(* Logix 5000 project; controller AMANA_DC_PLANT_01 vendor 1 type 14 code 164 rev 31.12; software revision 31.02 *)

TASK MainTask (continuous, watchdog 500 ms) : LN00, OH_BARCODE_SCAN

MODULES
   Local : vendor 1 type 14 code 164 (ICP 0, rev 31.12)
      EN4TR : 1756-EN4TR (ICP 3, Ethernet 192.168.1.1, rev 2.1, Input RPI 500 ms)
         Test_ArmorBlock : vendor 1 type 7 code 357 (Ethernet 192.168.1.100, rev 1.1, Output RPI 20 ms)
      OH_SCAN_DOCKSORTING : SR-2000 (Ethernet 10.28.17.144, rev 1.1, StandardDataDriven RPI 20 ms)
           OH_SCAN_DOCKSORTING:I.Data[0].0   // Error
           OH_SCAN_DOCKSORTING:I.Data[0].1   // Result Data Available
           OH_SCAN_DOCKSORTING:I.Data[0].2   // Result Data Strobe
           OH_SCAN_DOCKSORTING:I.Data[0].3   // Reserved
           OH_SCAN_DOCKSORTING:I.Data[0].4   // Reserved
           OH_SCAN_DOCKSORTING:I.Data[0].5   // Reserved
           OH_SCAN_DOCKSORTING:I.Data[0].6   // Buffer Overflow Error
           OH_SCAN_DOCKSORTING:I.Data[0].7   // General Error
           OH_SCAN_DOCKSORTING:I.Data[10]   // ISO/IEC15415 Grade
           OH_SCAN_DOCKSORTING:I.Data[11]   // Reserved
           OH_SCAN_DOCKSORTING:I.Data[12]   // AIM DPM Grade
           OH_SCAN_DOCKSORTING:I.Data[13]   // Reserved
           OH_SCAN_DOCKSORTING:I.Data[14]   // ISO/IEC15416 Grade
           OH_SCAN_DOCKSORTING:I.Data[15]   // Reserved
           OH_SCAN_DOCKSORTING:I.Data[16]   // Read Result Code
           OH_SCAN_DOCKSORTING:I.Data[17]   // Read Result Code
           OH_SCAN_DOCKSORTING:I.Data[18]   // Preset Result Code
           OH_SCAN_DOCKSORTING:I.Data[19]   // Preset Result Code
           OH_SCAN_DOCKSORTING:I.Data[1].0   // Busy
           OH_SCAN_DOCKSORTING:I.Data[1].1   // Trigger Busy
           OH_SCAN_DOCKSORTING:I.Data[1].2   // Lock Busy
           OH_SCAN_DOCKSORTING:I.Data[1].3   // Mode Busy
           OH_SCAN_DOCKSORTING:I.Data[1].4   // Error Busy
           OH_SCAN_DOCKSORTING:I.Data[1].5   // Reserved
           OH_SCAN_DOCKSORTING:I.Data[1].6   // Ready
           OH_SCAN_DOCKSORTING:I.Data[1].7   // Reserved
           OH_SCAN_DOCKSORTING:I.Data[20]   // Register Preset Data Result Code
           OH_SCAN_DOCKSORTING:I.Data[21]   // Register Preset Data Result Code
           OH_SCAN_DOCKSORTING:I.Data[22]   // Tune Result Code
           OH_SCAN_DOCKSORTING:I.Data[23]   // Tune Result Code
           OH_SCAN_DOCKSORTING:I.Data[24]   // Bload Result Code
           OH_SCAN_DOCKSORTING:I.Data[25]   // Bload Result Code
           OH_SCAN_DOCKSORTING:I.Data[26]   // Reserved
           OH_SCAN_DOCKSORTING:I.Data[27]   // Reserved
           OH_SCAN_DOCKSORTING:I.Data[28]   // Reserved
           OH_SCAN_DOCKSORTING:I.Data[29]   // Reserved
           OH_SCAN_DOCKSORTING:I.Data[2].0   // Read Complete
           OH_SCAN_DOCKSORTING:I.Data[2].1   // Preset Complete
           OH_SCAN_DOCKSORTING:I.Data[2].2   // Register Preset Data Complete
           OH_SCAN_DOCKSORTING:I.Data[2].3   // Tune Complete
           OH_SCAN_DOCKSORTING:I.Data[2].4   // Bload Complete
           OH_SCAN_DOCKSORTING:I.Data[2].5   // Reserved
           OH_SCAN_DOCKSORTING:I.Data[2].6   // Reserved
           OH_SCAN_DOCKSORTING:I.Data[2].7   // External Request Complete
           OH_SCAN_DOCKSORTING:I.Data[30]   // External Request Result Code
           OH_SCAN_DOCKSORTING:I.Data[31]   // External Request Result Code
           OH_SCAN_DOCKSORTING:I.Data[32]   // General Error Code
           OH_SCAN_DOCKSORTING:I.Data[33]   // General Error Code
           OH_SCAN_DOCKSORTING:I.Data[34]   // Slave ID
           OH_SCAN_DOCKSORTING:I.Data[35]   // Slave ID
           OH_SCAN_DOCKSORTING:I.Data[36]   // Result Data Ready Count
           OH_SCAN_DOCKSORTING:I.Data[37]   // Result Data Ready Count
           OH_SCAN_DOCKSORTING:I.Data[38]   // Result Data Update Count
           OH_SCAN_DOCKSORTING:I.Data[39]   // Result Data Update Count
           OH_SCAN_DOCKSORTING:I.Data[3].0   // Read Failure
           OH_SCAN_DOCKSORTING:I.Data[3].1   // Preset Failure
           OH_SCAN_DOCKSORTING:I.Data[3].2   // Register Preset Data Failure
           OH_SCAN_DOCKSORTING:I.Data[3].3   // Tune Failure
           OH_SCAN_DOCKSORTING:I.Data[3].4   // Bload Failure
           OH_SCAN_DOCKSORTING:I.Data[3].5   // Reserved
           OH_SCAN_DOCKSORTING:I.Data[3].6   // Reserved
           OH_SCAN_DOCKSORTING:I.Data[3].7   // External Request Failure
           OH_SCAN_DOCKSORTING:I.Data[40]   // Trigger Input Count for Master
           OH_SCAN_DOCKSORTING:I.Data[41]   // Trigger Input Count for Master
           OH_SCAN_DOCKSORTING:I.Data[42]   // Result Data Size
           OH_SCAN_DOCKSORTING:I.Data[43]   // Result Data Size
           OH_SCAN_DOCKSORTING:I.Data[44]   // Result Data
           OH_SCAN_DOCKSORTING:I.Data[45]   // Result Data
           OH_SCAN_DOCKSORTING:I.Data[46]   // Result Data
           OH_SCAN_DOCKSORTING:I.Data[47]   // Result Data
           OH_SCAN_DOCKSORTING:I.Data[48]   // Result Data
           OH_SCAN_DOCKSORTING:I.Data[49]   // Result Data
           OH_SCAN_DOCKSORTING:I.Data[4].0   // Input 1 Status
           OH_SCAN_DOCKSORTING:I.Data[4].1   // Input 2 Status
           OH_SCAN_DOCKSORTING:I.Data[4].2   // Reserved
           OH_SCAN_DOCKSORTING:I.Data[4].3   // Reserved
           OH_SCAN_DOCKSORTING:I.Data[4].4   // Output 1 Status
           OH_SCAN_DOCKSORTING:I.Data[4].5   // Output 2 Status
           OH_SCAN_DOCKSORTING:I.Data[4].6   // Output 3 Status
           OH_SCAN_DOCKSORTING:I.Data[4].7   // Reserved
           OH_SCAN_DOCKSORTING:I.Data[50]   // Result Data
           OH_SCAN_DOCKSORTING:I.Data[5].0   // Unstable
           OH_SCAN_DOCKSORTING:I.Data[5].1   // Matching Level Unstable
           OH_SCAN_DOCKSORTING:I.Data[5].2   // ISO/IEC15415 Unstable
           OH_SCAN_DOCKSORTING:I.Data[5].3   // AIM DPM Unstable
           OH_SCAN_DOCKSORTING:I.Data[5].4   // ADE AS9132 Unstable
           OH_SCAN_DOCKSORTING:I.Data[5].5   // ISO/IEC15416 Unstable
           OH_SCAN_DOCKSORTING:I.Data[5].6   // Reserved
           OH_SCAN_DOCKSORTING:I.Data[5].7   // Reserved
           OH_SCAN_DOCKSORTING:I.Data[6]   // Reserved
           OH_SCAN_DOCKSORTING:I.Data[7]   // Reserved
           OH_SCAN_DOCKSORTING:I.Data[8]   // Matching Level
           OH_SCAN_DOCKSORTING:I.Data[9]   // Reserved
           OH_SCAN_DOCKSORTING:O.Data[0].0   // Reserved
           OH_SCAN_DOCKSORTING:O.Data[0].1   // Result Data Latch
           OH_SCAN_DOCKSORTING:O.Data[0].2   // Reserved
           OH_SCAN_DOCKSORTING:O.Data[0].3   // Reserved
           OH_SCAN_DOCKSORTING:O.Data[0].4   // Reserved
           OH_SCAN_DOCKSORTING:O.Data[0].5   // Reserved
           OH_SCAN_DOCKSORTING:O.Data[0].6   // Reserved
           OH_SCAN_DOCKSORTING:O.Data[0].7   // Error Clear
           OH_SCAN_DOCKSORTING:O.Data[10]   // User Data Size
           OH_SCAN_DOCKSORTING:O.Data[11]   // User Data Size
           OH_SCAN_DOCKSORTING:O.Data[12]   // User Data
           OH_SCAN_DOCKSORTING:O.Data[13]   // User Data
           OH_SCAN_DOCKSORTING:O.Data[14]   // User Data
           OH_SCAN_DOCKSORTING:O.Data[15]   // User Data
           OH_SCAN_DOCKSORTING:O.Data[16]   // User Data
           OH_SCAN_DOCKSORTING:O.Data[17]   // User Data
           OH_SCAN_DOCKSORTING:O.Data[1].0   // Read Request
           OH_SCAN_DOCKSORTING:O.Data[1].1   // Preset Request
           OH_SCAN_DOCKSORTING:O.Data[1].2   // Register Preset Data Request
           OH_SCAN_DOCKSORTING:O.Data[1].3   // Tune Request
           OH_SCAN_DOCKSORTING:O.Data[1].4   // Bload Request
           OH_SCAN_DOCKSORTING:O.Data[1].5   // Reserved
           OH_SCAN_DOCKSORTING:O.Data[1].6   // Reserved
           OH_SCAN_DOCKSORTING:O.Data[1].7   // Reserved
           OH_SCAN_DOCKSORTING:O.Data[2].0   // Read Complete Clear
           OH_SCAN_DOCKSORTING:O.Data[2].1   // Preset Complete Clear
           OH_SCAN_DOCKSORTING:O.Data[2].2   // Register Preset Data Complete Clear
           OH_SCAN_DOCKSORTING:O.Data[2].3   // Tune Complete Clear
           OH_SCAN_DOCKSORTING:O.Data[2].4   // Bload Complete Clear
           OH_SCAN_DOCKSORTING:O.Data[2].5   // Reserved
           OH_SCAN_DOCKSORTING:O.Data[2].6   // Reserved
           OH_SCAN_DOCKSORTING:O.Data[2].7   // External Request Complete Clear
           OH_SCAN_DOCKSORTING:O.Data[3]   // Reserved
           OH_SCAN_DOCKSORTING:O.Data[4]   // Bank Number
           OH_SCAN_DOCKSORTING:O.Data[5]   // Bank Number
           OH_SCAN_DOCKSORTING:O.Data[6]   // Reserved
           OH_SCAN_DOCKSORTING:O.Data[7]   // Reserved
           OH_SCAN_DOCKSORTING:O.Data[8]   // Reserved
           OH_SCAN_DOCKSORTING:O.Data[9]   // Reserved
      OH_SCAN_WAREHOUSENORTH : SR-2000 (Ethernet 10.28.17.138, rev 1.1, StandardDataDriven RPI 20 ms)
           OH_SCAN_WAREHOUSENORTH:I.Data[0].0   // Error
           OH_SCAN_WAREHOUSENORTH:I.Data[0].1   // Result Data Available
           OH_SCAN_WAREHOUSENORTH:I.Data[0].2   // Result Data Strobe
           OH_SCAN_WAREHOUSENORTH:I.Data[0].3   // Reserved
           OH_SCAN_WAREHOUSENORTH:I.Data[0].4   // Reserved
           OH_SCAN_WAREHOUSENORTH:I.Data[0].5   // Reserved
           OH_SCAN_WAREHOUSENORTH:I.Data[0].6   // Buffer Overflow Error
           OH_SCAN_WAREHOUSENORTH:I.Data[0].7   // General Error
           OH_SCAN_WAREHOUSENORTH:I.Data[10]   // ISO/IEC15415 Grade
           OH_SCAN_WAREHOUSENORTH:I.Data[11]   // Reserved
           OH_SCAN_WAREHOUSENORTH:I.Data[12]   // AIM DPM Grade
           OH_SCAN_WAREHOUSENORTH:I.Data[13]   // Reserved
           OH_SCAN_WAREHOUSENORTH:I.Data[14]   // ISO/IEC15416 Grade
           OH_SCAN_WAREHOUSENORTH:I.Data[15]   // Reserved
           OH_SCAN_WAREHOUSENORTH:I.Data[16]   // Read Result Code
           OH_SCAN_WAREHOUSENORTH:I.Data[17]   // Read Result Code
           OH_SCAN_WAREHOUSENORTH:I.Data[18]   // Preset Result Code
           OH_SCAN_WAREHOUSENORTH:I.Data[19]   // Preset Result Code
           OH_SCAN_WAREHOUSENORTH:I.Data[1].0   // Busy
           OH_SCAN_WAREHOUSENORTH:I.Data[1].1   // Trigger Busy
           OH_SCAN_WAREHOUSENORTH:I.Data[1].2   // Lock Busy
           OH_SCAN_WAREHOUSENORTH:I.Data[1].3   // Mode Busy
           OH_SCAN_WAREHOUSENORTH:I.Data[1].4   // Error Busy
           OH_SCAN_WAREHOUSENORTH:I.Data[1].5   // Reserved
           OH_SCAN_WAREHOUSENORTH:I.Data[1].6   // Ready
           OH_SCAN_WAREHOUSENORTH:I.Data[1].7   // Reserved
           OH_SCAN_WAREHOUSENORTH:I.Data[20]   // Register Preset Data Result Code
           OH_SCAN_WAREHOUSENORTH:I.Data[21]   // Register Preset Data Result Code
           OH_SCAN_WAREHOUSENORTH:I.Data[22]   // Tune Result Code
           OH_SCAN_WAREHOUSENORTH:I.Data[23]   // Tune Result Code
           OH_SCAN_WAREHOUSENORTH:I.Data[24]   // Bload Result Code
           OH_SCAN_WAREHOUSENORTH:I.Data[25]   // Bload Result Code
           OH_SCAN_WAREHOUSENORTH:I.Data[26]   // Reserved
           OH_SCAN_WAREHOUSENORTH:I.Data[27]   // Reserved
           OH_SCAN_WAREHOUSENORTH:I.Data[28]   // Reserved
           OH_SCAN_WAREHOUSENORTH:I.Data[29]   // Reserved
           OH_SCAN_WAREHOUSENORTH:I.Data[2].0   // Read Complete
           OH_SCAN_WAREHOUSENORTH:I.Data[2].1   // Preset Complete
           OH_SCAN_WAREHOUSENORTH:I.Data[2].2   // Register Preset Data Complete
           OH_SCAN_WAREHOUSENORTH:I.Data[2].3   // Tune Complete
           OH_SCAN_WAREHOUSENORTH:I.Data[2].4   // Bload Complete
           OH_SCAN_WAREHOUSENORTH:I.Data[2].5   // Reserved
           OH_SCAN_WAREHOUSENORTH:I.Data[2].6   // Reserved
           OH_SCAN_WAREHOUSENORTH:I.Data[2].7   // External Request Complete
           OH_SCAN_WAREHOUSENORTH:I.Data[30]   // External Request Result Code
           OH_SCAN_WAREHOUSENORTH:I.Data[31]   // External Request Result Code
           OH_SCAN_WAREHOUSENORTH:I.Data[32]   // General Error Code
           OH_SCAN_WAREHOUSENORTH:I.Data[33]   // General Error Code
           OH_SCAN_WAREHOUSENORTH:I.Data[34]   // Slave ID
           OH_SCAN_WAREHOUSENORTH:I.Data[35]   // Slave ID
           OH_SCAN_WAREHOUSENORTH:I.Data[36]   // Result Data Ready Count
           OH_SCAN_WAREHOUSENORTH:I.Data[37]   // Result Data Ready Count
           OH_SCAN_WAREHOUSENORTH:I.Data[38]   // Result Data Update Count
           OH_SCAN_WAREHOUSENORTH:I.Data[39]   // Result Data Update Count
           OH_SCAN_WAREHOUSENORTH:I.Data[3].0   // Read Failure
           OH_SCAN_WAREHOUSENORTH:I.Data[3].1   // Preset Failure
           OH_SCAN_WAREHOUSENORTH:I.Data[3].2   // Register Preset Data Failure
           OH_SCAN_WAREHOUSENORTH:I.Data[3].3   // Tune Failure
           OH_SCAN_WAREHOUSENORTH:I.Data[3].4   // Bload Failure
           OH_SCAN_WAREHOUSENORTH:I.Data[3].5   // Reserved
           OH_SCAN_WAREHOUSENORTH:I.Data[3].6   // Reserved
           OH_SCAN_WAREHOUSENORTH:I.Data[3].7   // External Request Failure
           OH_SCAN_WAREHOUSENORTH:I.Data[40]   // Trigger Input Count for Master
           OH_SCAN_WAREHOUSENORTH:I.Data[41]   // Trigger Input Count for Master
           OH_SCAN_WAREHOUSENORTH:I.Data[42]   // Result Data Size
           OH_SCAN_WAREHOUSENORTH:I.Data[43]   // Result Data Size
           OH_SCAN_WAREHOUSENORTH:I.Data[44]   // Result Data
           OH_SCAN_WAREHOUSENORTH:I.Data[45]   // Result Data
           OH_SCAN_WAREHOUSENORTH:I.Data[46]   // Result Data
           OH_SCAN_WAREHOUSENORTH:I.Data[47]   // Result Data
           OH_SCAN_WAREHOUSENORTH:I.Data[48]   // Result Data
           OH_SCAN_WAREHOUSENORTH:I.Data[49]   // Result Data
           OH_SCAN_WAREHOUSENORTH:I.Data[4].0   // Input 1 Status
           OH_SCAN_WAREHOUSENORTH:I.Data[4].1   // Input 2 Status
           OH_SCAN_WAREHOUSENORTH:I.Data[4].2   // Reserved
           OH_SCAN_WAREHOUSENORTH:I.Data[4].3   // Reserved
           OH_SCAN_WAREHOUSENORTH:I.Data[4].4   // Output 1 Status
           OH_SCAN_WAREHOUSENORTH:I.Data[4].5   // Output 2 Status
           OH_SCAN_WAREHOUSENORTH:I.Data[4].6   // Output 3 Status
           OH_SCAN_WAREHOUSENORTH:I.Data[4].7   // Reserved
           OH_SCAN_WAREHOUSENORTH:I.Data[50]   // Result Data
           OH_SCAN_WAREHOUSENORTH:I.Data[5].0   // Unstable
           OH_SCAN_WAREHOUSENORTH:I.Data[5].1   // Matching Level Unstable
           OH_SCAN_WAREHOUSENORTH:I.Data[5].2   // ISO/IEC15415 Unstable
           OH_SCAN_WAREHOUSENORTH:I.Data[5].3   // AIM DPM Unstable
           OH_SCAN_WAREHOUSENORTH:I.Data[5].4   // ADE AS9132 Unstable
           OH_SCAN_WAREHOUSENORTH:I.Data[5].5   // ISO/IEC15416 Unstable
           OH_SCAN_WAREHOUSENORTH:I.Data[5].6   // Reserved
           OH_SCAN_WAREHOUSENORTH:I.Data[5].7   // Reserved
           OH_SCAN_WAREHOUSENORTH:I.Data[6]   // Reserved
           OH_SCAN_WAREHOUSENORTH:I.Data[7]   // Reserved
           OH_SCAN_WAREHOUSENORTH:I.Data[8]   // Matching Level
           OH_SCAN_WAREHOUSENORTH:I.Data[9]   // Reserved
           OH_SCAN_WAREHOUSENORTH:O.Data[0].0   // Reserved
           OH_SCAN_WAREHOUSENORTH:O.Data[0].1   // Result Data Latch
           OH_SCAN_WAREHOUSENORTH:O.Data[0].2   // Reserved
           OH_SCAN_WAREHOUSENORTH:O.Data[0].3   // Reserved
           OH_SCAN_WAREHOUSENORTH:O.Data[0].4   // Reserved
           OH_SCAN_WAREHOUSENORTH:O.Data[0].5   // Reserved
           OH_SCAN_WAREHOUSENORTH:O.Data[0].6   // Reserved
           OH_SCAN_WAREHOUSENORTH:O.Data[0].7   // Error Clear
           OH_SCAN_WAREHOUSENORTH:O.Data[10]   // User Data Size
           OH_SCAN_WAREHOUSENORTH:O.Data[11]   // User Data Size
           OH_SCAN_WAREHOUSENORTH:O.Data[12]   // User Data
           OH_SCAN_WAREHOUSENORTH:O.Data[13]   // User Data
           OH_SCAN_WAREHOUSENORTH:O.Data[14]   // User Data
           OH_SCAN_WAREHOUSENORTH:O.Data[15]   // User Data
           OH_SCAN_WAREHOUSENORTH:O.Data[16]   // User Data
           OH_SCAN_WAREHOUSENORTH:O.Data[17]   // User Data
           OH_SCAN_WAREHOUSENORTH:O.Data[1].0   // Read Request
           OH_SCAN_WAREHOUSENORTH:O.Data[1].1   // Preset Request
           OH_SCAN_WAREHOUSENORTH:O.Data[1].2   // Register Preset Data Request
           OH_SCAN_WAREHOUSENORTH:O.Data[1].3   // Tune Request
           OH_SCAN_WAREHOUSENORTH:O.Data[1].4   // Bload Request
           OH_SCAN_WAREHOUSENORTH:O.Data[1].5   // Reserved
           OH_SCAN_WAREHOUSENORTH:O.Data[1].6   // Reserved
           OH_SCAN_WAREHOUSENORTH:O.Data[1].7   // Reserved
           OH_SCAN_WAREHOUSENORTH:O.Data[2].0   // Read Complete Clear
           OH_SCAN_WAREHOUSENORTH:O.Data[2].1   // Preset Complete Clear
           OH_SCAN_WAREHOUSENORTH:O.Data[2].2   // Register Preset Data Complete Clear
           OH_SCAN_WAREHOUSENORTH:O.Data[2].3   // Tune Complete Clear
           OH_SCAN_WAREHOUSENORTH:O.Data[2].4   // Bload Complete Clear
           OH_SCAN_WAREHOUSENORTH:O.Data[2].5   // Reserved
           OH_SCAN_WAREHOUSENORTH:O.Data[2].6   // Reserved
           OH_SCAN_WAREHOUSENORTH:O.Data[2].7   // External Request Complete Clear
           OH_SCAN_WAREHOUSENORTH:O.Data[3]   // Reserved
           OH_SCAN_WAREHOUSENORTH:O.Data[4]   // Bank Number
           OH_SCAN_WAREHOUSENORTH:O.Data[5]   // Bank Number
           OH_SCAN_WAREHOUSENORTH:O.Data[6]   // Reserved
           OH_SCAN_WAREHOUSENORTH:O.Data[7]   // Reserved
           OH_SCAN_WAREHOUSENORTH:O.Data[8]   // Reserved
           OH_SCAN_WAREHOUSENORTH:O.Data[9]   // Reserved
      OH_SCAN_LN6 : SR-2000 (Ethernet 10.28.114.160, rev 1.1, StandardDataDriven RPI 20 ms)
           OH_SCAN_LN6:I.Data[0].0   // Error
           OH_SCAN_LN6:I.Data[0].1   // Result Data Available
           OH_SCAN_LN6:I.Data[0].2   // Result Data Strobe
           OH_SCAN_LN6:I.Data[0].3   // Reserved
           OH_SCAN_LN6:I.Data[0].4   // Reserved
           OH_SCAN_LN6:I.Data[0].5   // Reserved
           OH_SCAN_LN6:I.Data[0].6   // Buffer Overflow Error
           OH_SCAN_LN6:I.Data[0].7   // General Error
           OH_SCAN_LN6:I.Data[10]   // ISO/IEC15415 Grade
           OH_SCAN_LN6:I.Data[11]   // Reserved
           OH_SCAN_LN6:I.Data[12]   // AIM DPM Grade
           OH_SCAN_LN6:I.Data[13]   // Reserved
           OH_SCAN_LN6:I.Data[14]   // ISO/IEC15416 Grade
           OH_SCAN_LN6:I.Data[15]   // Reserved
           OH_SCAN_LN6:I.Data[16]   // Read Result Code
           OH_SCAN_LN6:I.Data[17]   // Read Result Code
           OH_SCAN_LN6:I.Data[18]   // Preset Result Code
           OH_SCAN_LN6:I.Data[19]   // Preset Result Code
           OH_SCAN_LN6:I.Data[1].0   // Busy
           OH_SCAN_LN6:I.Data[1].1   // Trigger Busy
           OH_SCAN_LN6:I.Data[1].2   // Lock Busy
           OH_SCAN_LN6:I.Data[1].3   // Mode Busy
           OH_SCAN_LN6:I.Data[1].4   // Error Busy
           OH_SCAN_LN6:I.Data[1].5   // Reserved
           OH_SCAN_LN6:I.Data[1].6   // Ready
           OH_SCAN_LN6:I.Data[1].7   // Reserved
           OH_SCAN_LN6:I.Data[20]   // Register Preset Data Result Code
           OH_SCAN_LN6:I.Data[21]   // Register Preset Data Result Code
           OH_SCAN_LN6:I.Data[22]   // Tune Result Code
           OH_SCAN_LN6:I.Data[23]   // Tune Result Code
           OH_SCAN_LN6:I.Data[24]   // Bload Result Code
           OH_SCAN_LN6:I.Data[25]   // Bload Result Code
           OH_SCAN_LN6:I.Data[26]   // Reserved
           OH_SCAN_LN6:I.Data[27]   // Reserved
           OH_SCAN_LN6:I.Data[28]   // Reserved
           OH_SCAN_LN6:I.Data[29]   // Reserved
           OH_SCAN_LN6:I.Data[2].0   // Read Complete
           OH_SCAN_LN6:I.Data[2].1   // Preset Complete
           OH_SCAN_LN6:I.Data[2].2   // Register Preset Data Complete
           OH_SCAN_LN6:I.Data[2].3   // Tune Complete
           OH_SCAN_LN6:I.Data[2].4   // Bload Complete
           OH_SCAN_LN6:I.Data[2].5   // Reserved
           OH_SCAN_LN6:I.Data[2].6   // Reserved
           OH_SCAN_LN6:I.Data[2].7   // External Request Complete
           OH_SCAN_LN6:I.Data[30]   // External Request Result Code
           OH_SCAN_LN6:I.Data[31]   // External Request Result Code
           OH_SCAN_LN6:I.Data[32]   // General Error Code
           OH_SCAN_LN6:I.Data[33]   // General Error Code
           OH_SCAN_LN6:I.Data[34]   // Slave ID
           OH_SCAN_LN6:I.Data[35]   // Slave ID
           OH_SCAN_LN6:I.Data[36]   // Result Data Ready Count
           OH_SCAN_LN6:I.Data[37]   // Result Data Ready Count
           OH_SCAN_LN6:I.Data[38]   // Result Data Update Count
           OH_SCAN_LN6:I.Data[39]   // Result Data Update Count
           OH_SCAN_LN6:I.Data[3].0   // Read Failure
           OH_SCAN_LN6:I.Data[3].1   // Preset Failure
           OH_SCAN_LN6:I.Data[3].2   // Register Preset Data Failure
           OH_SCAN_LN6:I.Data[3].3   // Tune Failure
           OH_SCAN_LN6:I.Data[3].4   // Bload Failure
           OH_SCAN_LN6:I.Data[3].5   // Reserved
           OH_SCAN_LN6:I.Data[3].6   // Reserved
           OH_SCAN_LN6:I.Data[3].7   // External Request Failure
           OH_SCAN_LN6:I.Data[40]   // Trigger Input Count for Master
           OH_SCAN_LN6:I.Data[41]   // Trigger Input Count for Master
           OH_SCAN_LN6:I.Data[42]   // Result Data Size
           OH_SCAN_LN6:I.Data[43]   // Result Data Size
           OH_SCAN_LN6:I.Data[44]   // Result Data
           OH_SCAN_LN6:I.Data[45]   // Result Data
           OH_SCAN_LN6:I.Data[46]   // Result Data
           OH_SCAN_LN6:I.Data[47]   // Result Data
           OH_SCAN_LN6:I.Data[48]   // Result Data
           OH_SCAN_LN6:I.Data[49]   // Result Data
           OH_SCAN_LN6:I.Data[4].0   // Input 1 Status
           OH_SCAN_LN6:I.Data[4].1   // Input 2 Status
           OH_SCAN_LN6:I.Data[4].2   // Reserved
           OH_SCAN_LN6:I.Data[4].3   // Reserved
           OH_SCAN_LN6:I.Data[4].4   // Output 1 Status
           OH_SCAN_LN6:I.Data[4].5   // Output 2 Status
           OH_SCAN_LN6:I.Data[4].6   // Output 3 Status
           OH_SCAN_LN6:I.Data[4].7   // Reserved
           OH_SCAN_LN6:I.Data[50]   // Result Data
           OH_SCAN_LN6:I.Data[5].0   // Unstable
           OH_SCAN_LN6:I.Data[5].1   // Matching Level Unstable
           OH_SCAN_LN6:I.Data[5].2   // ISO/IEC15415 Unstable
           OH_SCAN_LN6:I.Data[5].3   // AIM DPM Unstable
           OH_SCAN_LN6:I.Data[5].4   // ADE AS9132 Unstable
           OH_SCAN_LN6:I.Data[5].5   // ISO/IEC15416 Unstable
           OH_SCAN_LN6:I.Data[5].6   // Reserved
           OH_SCAN_LN6:I.Data[5].7   // Reserved
           OH_SCAN_LN6:I.Data[6]   // Reserved
           OH_SCAN_LN6:I.Data[7]   // Reserved
           OH_SCAN_LN6:I.Data[8]   // Matching Level
           OH_SCAN_LN6:I.Data[9]   // Reserved
           OH_SCAN_LN6:O.Data[0].0   // Reserved
           OH_SCAN_LN6:O.Data[0].1   // Result Data Latch
           OH_SCAN_LN6:O.Data[0].2   // Reserved
           OH_SCAN_LN6:O.Data[0].3   // Reserved
           OH_SCAN_LN6:O.Data[0].4   // Reserved
           OH_SCAN_LN6:O.Data[0].5   // Reserved
           OH_SCAN_LN6:O.Data[0].6   // Reserved
           OH_SCAN_LN6:O.Data[0].7   // Error Clear
           OH_SCAN_LN6:O.Data[10]   // User Data Size
           OH_SCAN_LN6:O.Data[11]   // User Data Size
           OH_SCAN_LN6:O.Data[12]   // User Data
           OH_SCAN_LN6:O.Data[13]   // User Data
           OH_SCAN_LN6:O.Data[14]   // User Data
           OH_SCAN_LN6:O.Data[15]   // User Data
           OH_SCAN_LN6:O.Data[16]   // User Data
           OH_SCAN_LN6:O.Data[17]   // User Data
           OH_SCAN_LN6:O.Data[1].0   // Read Request
           OH_SCAN_LN6:O.Data[1].1   // Preset Request
           OH_SCAN_LN6:O.Data[1].2   // Register Preset Data Request
           OH_SCAN_LN6:O.Data[1].3   // Tune Request
           OH_SCAN_LN6:O.Data[1].4   // Bload Request
           OH_SCAN_LN6:O.Data[1].5   // Reserved
           OH_SCAN_LN6:O.Data[1].6   // Reserved
           OH_SCAN_LN6:O.Data[1].7   // Reserved
           OH_SCAN_LN6:O.Data[2].0   // Read Complete Clear
           OH_SCAN_LN6:O.Data[2].1   // Preset Complete Clear
           OH_SCAN_LN6:O.Data[2].2   // Register Preset Data Complete Clear
           OH_SCAN_LN6:O.Data[2].3   // Tune Complete Clear
           OH_SCAN_LN6:O.Data[2].4   // Bload Complete Clear
           OH_SCAN_LN6:O.Data[2].5   // Reserved
           OH_SCAN_LN6:O.Data[2].6   // Reserved
           OH_SCAN_LN6:O.Data[2].7   // External Request Complete Clear
           OH_SCAN_LN6:O.Data[3]   // Reserved
           OH_SCAN_LN6:O.Data[4]   // Bank Number
           OH_SCAN_LN6:O.Data[5]   // Bank Number
           OH_SCAN_LN6:O.Data[6]   // Reserved
           OH_SCAN_LN6:O.Data[7]   // Reserved
           OH_SCAN_LN6:O.Data[8]   // Reserved
           OH_SCAN_LN6:O.Data[9]   // Reserved
      OH_SCAN_LN67MERGE : SR-2000 (Ethernet 10.28.64.200, rev 1.1, StandardDataDriven RPI 20 ms)
           OH_SCAN_LN67MERGE:I.Data[0].0   // Error
           OH_SCAN_LN67MERGE:I.Data[0].1   // Result Data Available
           OH_SCAN_LN67MERGE:I.Data[0].2   // Result Data Strobe
           OH_SCAN_LN67MERGE:I.Data[0].3   // Reserved
           OH_SCAN_LN67MERGE:I.Data[0].4   // Reserved
           OH_SCAN_LN67MERGE:I.Data[0].5   // Reserved
           OH_SCAN_LN67MERGE:I.Data[0].6   // Buffer Overflow Error
           OH_SCAN_LN67MERGE:I.Data[0].7   // General Error
           OH_SCAN_LN67MERGE:I.Data[10]   // ISO/IEC15415 Grade
           OH_SCAN_LN67MERGE:I.Data[11]   // Reserved
           OH_SCAN_LN67MERGE:I.Data[12]   // AIM DPM Grade
           OH_SCAN_LN67MERGE:I.Data[13]   // Reserved
           OH_SCAN_LN67MERGE:I.Data[14]   // ISO/IEC15416 Grade
           OH_SCAN_LN67MERGE:I.Data[15]   // Reserved
           OH_SCAN_LN67MERGE:I.Data[16]   // Read Result Code
           OH_SCAN_LN67MERGE:I.Data[17]   // Read Result Code
           OH_SCAN_LN67MERGE:I.Data[18]   // Preset Result Code
           OH_SCAN_LN67MERGE:I.Data[19]   // Preset Result Code
           OH_SCAN_LN67MERGE:I.Data[1].0   // Busy
           OH_SCAN_LN67MERGE:I.Data[1].1   // Trigger Busy
           OH_SCAN_LN67MERGE:I.Data[1].2   // Lock Busy
           OH_SCAN_LN67MERGE:I.Data[1].3   // Mode Busy
           OH_SCAN_LN67MERGE:I.Data[1].4   // Error Busy
           OH_SCAN_LN67MERGE:I.Data[1].5   // Reserved
           OH_SCAN_LN67MERGE:I.Data[1].6   // Ready
           OH_SCAN_LN67MERGE:I.Data[1].7   // Reserved
           OH_SCAN_LN67MERGE:I.Data[20]   // Register Preset Data Result Code
           OH_SCAN_LN67MERGE:I.Data[21]   // Register Preset Data Result Code
           OH_SCAN_LN67MERGE:I.Data[22]   // Tune Result Code
           OH_SCAN_LN67MERGE:I.Data[23]   // Tune Result Code
           OH_SCAN_LN67MERGE:I.Data[24]   // Bload Result Code
           OH_SCAN_LN67MERGE:I.Data[25]   // Bload Result Code
           OH_SCAN_LN67MERGE:I.Data[26]   // Reserved
           OH_SCAN_LN67MERGE:I.Data[27]   // Reserved
           OH_SCAN_LN67MERGE:I.Data[28]   // Reserved
           OH_SCAN_LN67MERGE:I.Data[29]   // Reserved
           OH_SCAN_LN67MERGE:I.Data[2].0   // Read Complete
           OH_SCAN_LN67MERGE:I.Data[2].1   // Preset Complete
           OH_SCAN_LN67MERGE:I.Data[2].2   // Register Preset Data Complete
           OH_SCAN_LN67MERGE:I.Data[2].3   // Tune Complete
           OH_SCAN_LN67MERGE:I.Data[2].4   // Bload Complete
           OH_SCAN_LN67MERGE:I.Data[2].5   // Reserved
           OH_SCAN_LN67MERGE:I.Data[2].6   // Reserved
           OH_SCAN_LN67MERGE:I.Data[2].7   // External Request Complete
           OH_SCAN_LN67MERGE:I.Data[30]   // External Request Result Code
           OH_SCAN_LN67MERGE:I.Data[31]   // External Request Result Code
           OH_SCAN_LN67MERGE:I.Data[32]   // General Error Code
           OH_SCAN_LN67MERGE:I.Data[33]   // General Error Code
           OH_SCAN_LN67MERGE:I.Data[34]   // Slave ID
           OH_SCAN_LN67MERGE:I.Data[35]   // Slave ID
           OH_SCAN_LN67MERGE:I.Data[36]   // Result Data Ready Count
           OH_SCAN_LN67MERGE:I.Data[37]   // Result Data Ready Count
           OH_SCAN_LN67MERGE:I.Data[38]   // Result Data Update Count
           OH_SCAN_LN67MERGE:I.Data[39]   // Result Data Update Count
           OH_SCAN_LN67MERGE:I.Data[3].0   // Read Failure
           OH_SCAN_LN67MERGE:I.Data[3].1   // Preset Failure
           OH_SCAN_LN67MERGE:I.Data[3].2   // Register Preset Data Failure
           OH_SCAN_LN67MERGE:I.Data[3].3   // Tune Failure
           OH_SCAN_LN67MERGE:I.Data[3].4   // Bload Failure
           OH_SCAN_LN67MERGE:I.Data[3].5   // Reserved
           OH_SCAN_LN67MERGE:I.Data[3].6   // Reserved
           OH_SCAN_LN67MERGE:I.Data[3].7   // External Request Failure
           OH_SCAN_LN67MERGE:I.Data[40]   // Trigger Input Count for Master
           OH_SCAN_LN67MERGE:I.Data[41]   // Trigger Input Count for Master
           OH_SCAN_LN67MERGE:I.Data[42]   // Result Data Size
           OH_SCAN_LN67MERGE:I.Data[43]   // Result Data Size
           OH_SCAN_LN67MERGE:I.Data[44]   // Result Data
           OH_SCAN_LN67MERGE:I.Data[45]   // Result Data
           OH_SCAN_LN67MERGE:I.Data[46]   // Result Data
           OH_SCAN_LN67MERGE:I.Data[47]   // Result Data
           OH_SCAN_LN67MERGE:I.Data[48]   // Result Data
           OH_SCAN_LN67MERGE:I.Data[49]   // Result Data
           OH_SCAN_LN67MERGE:I.Data[4].0   // Input 1 Status
           OH_SCAN_LN67MERGE:I.Data[4].1   // Input 2 Status
           OH_SCAN_LN67MERGE:I.Data[4].2   // Reserved
           OH_SCAN_LN67MERGE:I.Data[4].3   // Reserved
           OH_SCAN_LN67MERGE:I.Data[4].4   // Output 1 Status
           OH_SCAN_LN67MERGE:I.Data[4].5   // Output 2 Status
           OH_SCAN_LN67MERGE:I.Data[4].6   // Output 3 Status
           OH_SCAN_LN67MERGE:I.Data[4].7   // Reserved
           OH_SCAN_LN67MERGE:I.Data[50]   // Result Data
           OH_SCAN_LN67MERGE:I.Data[5].0   // Unstable
           OH_SCAN_LN67MERGE:I.Data[5].1   // Matching Level Unstable
           OH_SCAN_LN67MERGE:I.Data[5].2   // ISO/IEC15415 Unstable
           OH_SCAN_LN67MERGE:I.Data[5].3   // AIM DPM Unstable
           OH_SCAN_LN67MERGE:I.Data[5].4   // ADE AS9132 Unstable
           OH_SCAN_LN67MERGE:I.Data[5].5   // ISO/IEC15416 Unstable
           OH_SCAN_LN67MERGE:I.Data[5].6   // Reserved
           OH_SCAN_LN67MERGE:I.Data[5].7   // Reserved
           OH_SCAN_LN67MERGE:I.Data[6]   // Reserved
           OH_SCAN_LN67MERGE:I.Data[7]   // Reserved
           OH_SCAN_LN67MERGE:I.Data[8]   // Matching Level
           OH_SCAN_LN67MERGE:I.Data[9]   // Reserved
           OH_SCAN_LN67MERGE:O.Data[0].0   // Reserved
           OH_SCAN_LN67MERGE:O.Data[0].1   // Result Data Latch
           OH_SCAN_LN67MERGE:O.Data[0].2   // Reserved
           OH_SCAN_LN67MERGE:O.Data[0].3   // Reserved
           OH_SCAN_LN67MERGE:O.Data[0].4   // Reserved
           OH_SCAN_LN67MERGE:O.Data[0].5   // Reserved
           OH_SCAN_LN67MERGE:O.Data[0].6   // Reserved
           OH_SCAN_LN67MERGE:O.Data[0].7   // Error Clear
           OH_SCAN_LN67MERGE:O.Data[10]   // User Data Size
           OH_SCAN_LN67MERGE:O.Data[11]   // User Data Size
           OH_SCAN_LN67MERGE:O.Data[12]   // User Data
           OH_SCAN_LN67MERGE:O.Data[13]   // User Data
           OH_SCAN_LN67MERGE:O.Data[14]   // User Data
           OH_SCAN_LN67MERGE:O.Data[15]   // User Data
           OH_SCAN_LN67MERGE:O.Data[16]   // User Data
           OH_SCAN_LN67MERGE:O.Data[17]   // User Data
           OH_SCAN_LN67MERGE:O.Data[1].0   // Read Request
           OH_SCAN_LN67MERGE:O.Data[1].1   // Preset Request
           OH_SCAN_LN67MERGE:O.Data[1].2   // Register Preset Data Request
           OH_SCAN_LN67MERGE:O.Data[1].3   // Tune Request
           OH_SCAN_LN67MERGE:O.Data[1].4   // Bload Request
           OH_SCAN_LN67MERGE:O.Data[1].5   // Reserved
           OH_SCAN_LN67MERGE:O.Data[1].6   // Reserved
           OH_SCAN_LN67MERGE:O.Data[1].7   // Reserved
           OH_SCAN_LN67MERGE:O.Data[2].0   // Read Complete Clear
           OH_SCAN_LN67MERGE:O.Data[2].1   // Preset Complete Clear
           OH_SCAN_LN67MERGE:O.Data[2].2   // Register Preset Data Complete Clear
           OH_SCAN_LN67MERGE:O.Data[2].3   // Tune Complete Clear
           OH_SCAN_LN67MERGE:O.Data[2].4   // Bload Complete Clear
           OH_SCAN_LN67MERGE:O.Data[2].5   // Reserved
           OH_SCAN_LN67MERGE:O.Data[2].6   // Reserved
           OH_SCAN_LN67MERGE:O.Data[2].7   // External Request Complete Clear
           OH_SCAN_LN67MERGE:O.Data[3]   // Reserved
           OH_SCAN_LN67MERGE:O.Data[4]   // Bank Number
           OH_SCAN_LN67MERGE:O.Data[5]   // Bank Number
           OH_SCAN_LN67MERGE:O.Data[6]   // Reserved
           OH_SCAN_LN67MERGE:O.Data[7]   // Reserved
           OH_SCAN_LN67MERGE:O.Data[8]   // Reserved
           OH_SCAN_LN67MERGE:O.Data[9]   // Reserved
      OH_SCAN_LONGTERMEAST : SR-2000 (Ethernet 10.28.17.140, rev 1.1, StandardDataDriven RPI 20 ms)
           OH_SCAN_LONGTERMEAST:I.Data[0].0   // Error
           OH_SCAN_LONGTERMEAST:I.Data[0].1   // Result Data Available
           OH_SCAN_LONGTERMEAST:I.Data[0].2   // Result Data Strobe
           OH_SCAN_LONGTERMEAST:I.Data[0].3   // Reserved
           OH_SCAN_LONGTERMEAST:I.Data[0].4   // Reserved
           OH_SCAN_LONGTERMEAST:I.Data[0].5   // Reserved
           OH_SCAN_LONGTERMEAST:I.Data[0].6   // Buffer Overflow Error
           OH_SCAN_LONGTERMEAST:I.Data[0].7   // General Error
           OH_SCAN_LONGTERMEAST:I.Data[10]   // ISO/IEC15415 Grade
           OH_SCAN_LONGTERMEAST:I.Data[11]   // Reserved
           OH_SCAN_LONGTERMEAST:I.Data[12]   // AIM DPM Grade
           OH_SCAN_LONGTERMEAST:I.Data[13]   // Reserved
           OH_SCAN_LONGTERMEAST:I.Data[14]   // ISO/IEC15416 Grade
           OH_SCAN_LONGTERMEAST:I.Data[15]   // Reserved
           OH_SCAN_LONGTERMEAST:I.Data[16]   // Read Result Code
           OH_SCAN_LONGTERMEAST:I.Data[17]   // Read Result Code
           OH_SCAN_LONGTERMEAST:I.Data[18]   // Preset Result Code
           OH_SCAN_LONGTERMEAST:I.Data[19]   // Preset Result Code
           OH_SCAN_LONGTERMEAST:I.Data[1].0   // Busy
           OH_SCAN_LONGTERMEAST:I.Data[1].1   // Trigger Busy
           OH_SCAN_LONGTERMEAST:I.Data[1].2   // Lock Busy
           OH_SCAN_LONGTERMEAST:I.Data[1].3   // Mode Busy
           OH_SCAN_LONGTERMEAST:I.Data[1].4   // Error Busy
           OH_SCAN_LONGTERMEAST:I.Data[1].5   // Reserved
           OH_SCAN_LONGTERMEAST:I.Data[1].6   // Ready
           OH_SCAN_LONGTERMEAST:I.Data[1].7   // Reserved
           OH_SCAN_LONGTERMEAST:I.Data[20]   // Register Preset Data Result Code
           OH_SCAN_LONGTERMEAST:I.Data[21]   // Register Preset Data Result Code
           OH_SCAN_LONGTERMEAST:I.Data[22]   // Tune Result Code
           OH_SCAN_LONGTERMEAST:I.Data[23]   // Tune Result Code
           OH_SCAN_LONGTERMEAST:I.Data[24]   // Bload Result Code
           OH_SCAN_LONGTERMEAST:I.Data[25]   // Bload Result Code
           OH_SCAN_LONGTERMEAST:I.Data[26]   // Reserved
           OH_SCAN_LONGTERMEAST:I.Data[27]   // Reserved
           OH_SCAN_LONGTERMEAST:I.Data[28]   // Reserved
           OH_SCAN_LONGTERMEAST:I.Data[29]   // Reserved
           OH_SCAN_LONGTERMEAST:I.Data[2].0   // Read Complete
           OH_SCAN_LONGTERMEAST:I.Data[2].1   // Preset Complete
           OH_SCAN_LONGTERMEAST:I.Data[2].2   // Register Preset Data Complete
           OH_SCAN_LONGTERMEAST:I.Data[2].3   // Tune Complete
           OH_SCAN_LONGTERMEAST:I.Data[2].4   // Bload Complete
           OH_SCAN_LONGTERMEAST:I.Data[2].5   // Reserved
           OH_SCAN_LONGTERMEAST:I.Data[2].6   // Reserved
           OH_SCAN_LONGTERMEAST:I.Data[2].7   // External Request Complete
           OH_SCAN_LONGTERMEAST:I.Data[30]   // External Request Result Code
           OH_SCAN_LONGTERMEAST:I.Data[31]   // External Request Result Code
           OH_SCAN_LONGTERMEAST:I.Data[32]   // General Error Code
           OH_SCAN_LONGTERMEAST:I.Data[33]   // General Error Code
           OH_SCAN_LONGTERMEAST:I.Data[34]   // Slave ID
           OH_SCAN_LONGTERMEAST:I.Data[35]   // Slave ID
           OH_SCAN_LONGTERMEAST:I.Data[36]   // Result Data Ready Count
           OH_SCAN_LONGTERMEAST:I.Data[37]   // Result Data Ready Count
           OH_SCAN_LONGTERMEAST:I.Data[38]   // Result Data Update Count
           OH_SCAN_LONGTERMEAST:I.Data[39]   // Result Data Update Count
           OH_SCAN_LONGTERMEAST:I.Data[3].0   // Read Failure
           OH_SCAN_LONGTERMEAST:I.Data[3].1   // Preset Failure
           OH_SCAN_LONGTERMEAST:I.Data[3].2   // Register Preset Data Failure
           OH_SCAN_LONGTERMEAST:I.Data[3].3   // Tune Failure
           OH_SCAN_LONGTERMEAST:I.Data[3].4   // Bload Failure
           OH_SCAN_LONGTERMEAST:I.Data[3].5   // Reserved
           OH_SCAN_LONGTERMEAST:I.Data[3].6   // Reserved
           OH_SCAN_LONGTERMEAST:I.Data[3].7   // External Request Failure
           OH_SCAN_LONGTERMEAST:I.Data[40]   // Trigger Input Count for Master
           OH_SCAN_LONGTERMEAST:I.Data[41]   // Trigger Input Count for Master
           OH_SCAN_LONGTERMEAST:I.Data[42]   // Result Data Size
           OH_SCAN_LONGTERMEAST:I.Data[43]   // Result Data Size
           OH_SCAN_LONGTERMEAST:I.Data[44]   // Result Data
           OH_SCAN_LONGTERMEAST:I.Data[45]   // Result Data
           OH_SCAN_LONGTERMEAST:I.Data[46]   // Result Data
           OH_SCAN_LONGTERMEAST:I.Data[47]   // Result Data
           OH_SCAN_LONGTERMEAST:I.Data[48]   // Result Data
           OH_SCAN_LONGTERMEAST:I.Data[49]   // Result Data
           OH_SCAN_LONGTERMEAST:I.Data[4].0   // Input 1 Status
           OH_SCAN_LONGTERMEAST:I.Data[4].1   // Input 2 Status
           OH_SCAN_LONGTERMEAST:I.Data[4].2   // Reserved
           OH_SCAN_LONGTERMEAST:I.Data[4].3   // Reserved
           OH_SCAN_LONGTERMEAST:I.Data[4].4   // Output 1 Status
           OH_SCAN_LONGTERMEAST:I.Data[4].5   // Output 2 Status
           OH_SCAN_LONGTERMEAST:I.Data[4].6   // Output 3 Status
           OH_SCAN_LONGTERMEAST:I.Data[4].7   // Reserved
           OH_SCAN_LONGTERMEAST:I.Data[50]   // Result Data
           OH_SCAN_LONGTERMEAST:I.Data[5].0   // Unstable
           OH_SCAN_LONGTERMEAST:I.Data[5].1   // Matching Level Unstable
           OH_SCAN_LONGTERMEAST:I.Data[5].2   // ISO/IEC15415 Unstable
           OH_SCAN_LONGTERMEAST:I.Data[5].3   // AIM DPM Unstable
           OH_SCAN_LONGTERMEAST:I.Data[5].4   // ADE AS9132 Unstable
           OH_SCAN_LONGTERMEAST:I.Data[5].5   // ISO/IEC15416 Unstable
           OH_SCAN_LONGTERMEAST:I.Data[5].6   // Reserved
           OH_SCAN_LONGTERMEAST:I.Data[5].7   // Reserved
           OH_SCAN_LONGTERMEAST:I.Data[6]   // Reserved
           OH_SCAN_LONGTERMEAST:I.Data[7]   // Reserved
           OH_SCAN_LONGTERMEAST:I.Data[8]   // Matching Level
           OH_SCAN_LONGTERMEAST:I.Data[9]   // Reserved
           OH_SCAN_LONGTERMEAST:O.Data[0].0   // Reserved
           OH_SCAN_LONGTERMEAST:O.Data[0].1   // Result Data Latch
           OH_SCAN_LONGTERMEAST:O.Data[0].2   // Reserved
           OH_SCAN_LONGTERMEAST:O.Data[0].3   // Reserved
           OH_SCAN_LONGTERMEAST:O.Data[0].4   // Reserved
           OH_SCAN_LONGTERMEAST:O.Data[0].5   // Reserved
           OH_SCAN_LONGTERMEAST:O.Data[0].6   // Reserved
           OH_SCAN_LONGTERMEAST:O.Data[0].7   // Error Clear
           OH_SCAN_LONGTERMEAST:O.Data[10]   // User Data Size
           OH_SCAN_LONGTERMEAST:O.Data[11]   // User Data Size
           OH_SCAN_LONGTERMEAST:O.Data[12]   // User Data
           OH_SCAN_LONGTERMEAST:O.Data[13]   // User Data
           OH_SCAN_LONGTERMEAST:O.Data[14]   // User Data
           OH_SCAN_LONGTERMEAST:O.Data[15]   // User Data
           OH_SCAN_LONGTERMEAST:O.Data[16]   // User Data
           OH_SCAN_LONGTERMEAST:O.Data[17]   // User Data
           OH_SCAN_LONGTERMEAST:O.Data[1].0   // Read Request
           OH_SCAN_LONGTERMEAST:O.Data[1].1   // Preset Request
           OH_SCAN_LONGTERMEAST:O.Data[1].2   // Register Preset Data Request
           OH_SCAN_LONGTERMEAST:O.Data[1].3   // Tune Request
           OH_SCAN_LONGTERMEAST:O.Data[1].4   // Bload Request
           OH_SCAN_LONGTERMEAST:O.Data[1].5   // Reserved
           OH_SCAN_LONGTERMEAST:O.Data[1].6   // Reserved
           OH_SCAN_LONGTERMEAST:O.Data[1].7   // Reserved
           OH_SCAN_LONGTERMEAST:O.Data[2].0   // Read Complete Clear
           OH_SCAN_LONGTERMEAST:O.Data[2].1   // Preset Complete Clear
           OH_SCAN_LONGTERMEAST:O.Data[2].2   // Register Preset Data Complete Clear
           OH_SCAN_LONGTERMEAST:O.Data[2].3   // Tune Complete Clear
           OH_SCAN_LONGTERMEAST:O.Data[2].4   // Bload Complete Clear
           OH_SCAN_LONGTERMEAST:O.Data[2].5   // Reserved
           OH_SCAN_LONGTERMEAST:O.Data[2].6   // Reserved
           OH_SCAN_LONGTERMEAST:O.Data[2].7   // External Request Complete Clear
           OH_SCAN_LONGTERMEAST:O.Data[3]   // Reserved
           OH_SCAN_LONGTERMEAST:O.Data[4]   // Bank Number
           OH_SCAN_LONGTERMEAST:O.Data[5]   // Bank Number
           OH_SCAN_LONGTERMEAST:O.Data[6]   // Reserved
           OH_SCAN_LONGTERMEAST:O.Data[7]   // Reserved
           OH_SCAN_LONGTERMEAST:O.Data[8]   // Reserved
           OH_SCAN_LONGTERMEAST:O.Data[9]   // Reserved
      OH_SCAN_LN467MERGE : SR-2000 (Ethernet 10.28.17.142, rev 1.1, StandardDataDriven RPI 20 ms)
           OH_SCAN_LN467MERGE:I.Data[0].0   // Error
           OH_SCAN_LN467MERGE:I.Data[0].1   // Result Data Available
           OH_SCAN_LN467MERGE:I.Data[0].2   // Result Data Strobe
           OH_SCAN_LN467MERGE:I.Data[0].3   // Reserved
           OH_SCAN_LN467MERGE:I.Data[0].4   // Reserved
           OH_SCAN_LN467MERGE:I.Data[0].5   // Reserved
           OH_SCAN_LN467MERGE:I.Data[0].6   // Buffer Overflow Error
           OH_SCAN_LN467MERGE:I.Data[0].7   // General Error
           OH_SCAN_LN467MERGE:I.Data[10]   // ISO/IEC15415 Grade
           OH_SCAN_LN467MERGE:I.Data[11]   // Reserved
           OH_SCAN_LN467MERGE:I.Data[12]   // AIM DPM Grade
           OH_SCAN_LN467MERGE:I.Data[13]   // Reserved
           OH_SCAN_LN467MERGE:I.Data[14]   // ISO/IEC15416 Grade
           OH_SCAN_LN467MERGE:I.Data[15]   // Reserved
           OH_SCAN_LN467MERGE:I.Data[16]   // Read Result Code
           OH_SCAN_LN467MERGE:I.Data[17]   // Read Result Code
           OH_SCAN_LN467MERGE:I.Data[18]   // Preset Result Code
           OH_SCAN_LN467MERGE:I.Data[19]   // Preset Result Code
           OH_SCAN_LN467MERGE:I.Data[1].0   // Busy
           OH_SCAN_LN467MERGE:I.Data[1].1   // Trigger Busy
           OH_SCAN_LN467MERGE:I.Data[1].2   // Lock Busy
           OH_SCAN_LN467MERGE:I.Data[1].3   // Mode Busy
           OH_SCAN_LN467MERGE:I.Data[1].4   // Error Busy
           OH_SCAN_LN467MERGE:I.Data[1].5   // Reserved
           OH_SCAN_LN467MERGE:I.Data[1].6   // Ready
           OH_SCAN_LN467MERGE:I.Data[1].7   // Reserved
           OH_SCAN_LN467MERGE:I.Data[20]   // Register Preset Data Result Code
           OH_SCAN_LN467MERGE:I.Data[21]   // Register Preset Data Result Code
           OH_SCAN_LN467MERGE:I.Data[22]   // Tune Result Code
           OH_SCAN_LN467MERGE:I.Data[23]   // Tune Result Code
           OH_SCAN_LN467MERGE:I.Data[24]   // Bload Result Code
           OH_SCAN_LN467MERGE:I.Data[25]   // Bload Result Code
           OH_SCAN_LN467MERGE:I.Data[26]   // Reserved
           OH_SCAN_LN467MERGE:I.Data[27]   // Reserved
           OH_SCAN_LN467MERGE:I.Data[28]   // Reserved
           OH_SCAN_LN467MERGE:I.Data[29]   // Reserved
           OH_SCAN_LN467MERGE:I.Data[2].0   // Read Complete
           OH_SCAN_LN467MERGE:I.Data[2].1   // Preset Complete
           OH_SCAN_LN467MERGE:I.Data[2].2   // Register Preset Data Complete
           OH_SCAN_LN467MERGE:I.Data[2].3   // Tune Complete
           OH_SCAN_LN467MERGE:I.Data[2].4   // Bload Complete
           OH_SCAN_LN467MERGE:I.Data[2].5   // Reserved
           OH_SCAN_LN467MERGE:I.Data[2].6   // Reserved
           OH_SCAN_LN467MERGE:I.Data[2].7   // External Request Complete
           OH_SCAN_LN467MERGE:I.Data[30]   // External Request Result Code
           OH_SCAN_LN467MERGE:I.Data[31]   // External Request Result Code
           OH_SCAN_LN467MERGE:I.Data[32]   // General Error Code
           OH_SCAN_LN467MERGE:I.Data[33]   // General Error Code
           OH_SCAN_LN467MERGE:I.Data[34]   // Slave ID
           OH_SCAN_LN467MERGE:I.Data[35]   // Slave ID
           OH_SCAN_LN467MERGE:I.Data[36]   // Result Data Ready Count
           OH_SCAN_LN467MERGE:I.Data[37]   // Result Data Ready Count
           OH_SCAN_LN467MERGE:I.Data[38]   // Result Data Update Count
           OH_SCAN_LN467MERGE:I.Data[39]   // Result Data Update Count
           OH_SCAN_LN467MERGE:I.Data[3].0   // Read Failure
           OH_SCAN_LN467MERGE:I.Data[3].1   // Preset Failure
           OH_SCAN_LN467MERGE:I.Data[3].2   // Register Preset Data Failure
           OH_SCAN_LN467MERGE:I.Data[3].3   // Tune Failure
           OH_SCAN_LN467MERGE:I.Data[3].4   // Bload Failure
           OH_SCAN_LN467MERGE:I.Data[3].5   // Reserved
           OH_SCAN_LN467MERGE:I.Data[3].6   // Reserved
           OH_SCAN_LN467MERGE:I.Data[3].7   // External Request Failure
           OH_SCAN_LN467MERGE:I.Data[40]   // Trigger Input Count for Master
           OH_SCAN_LN467MERGE:I.Data[41]   // Trigger Input Count for Master
           OH_SCAN_LN467MERGE:I.Data[42]   // Result Data Size
           OH_SCAN_LN467MERGE:I.Data[43]   // Result Data Size
           OH_SCAN_LN467MERGE:I.Data[44]   // Result Data
           OH_SCAN_LN467MERGE:I.Data[45]   // Result Data
           OH_SCAN_LN467MERGE:I.Data[46]   // Result Data
           OH_SCAN_LN467MERGE:I.Data[47]   // Result Data
           OH_SCAN_LN467MERGE:I.Data[48]   // Result Data
           OH_SCAN_LN467MERGE:I.Data[49]   // Result Data
           OH_SCAN_LN467MERGE:I.Data[4].0   // Input 1 Status
           OH_SCAN_LN467MERGE:I.Data[4].1   // Input 2 Status
           OH_SCAN_LN467MERGE:I.Data[4].2   // Reserved
           OH_SCAN_LN467MERGE:I.Data[4].3   // Reserved
           OH_SCAN_LN467MERGE:I.Data[4].4   // Output 1 Status
           OH_SCAN_LN467MERGE:I.Data[4].5   // Output 2 Status
           OH_SCAN_LN467MERGE:I.Data[4].6   // Output 3 Status
           OH_SCAN_LN467MERGE:I.Data[4].7   // Reserved
           OH_SCAN_LN467MERGE:I.Data[50]   // Result Data
           OH_SCAN_LN467MERGE:I.Data[5].0   // Unstable
           OH_SCAN_LN467MERGE:I.Data[5].1   // Matching Level Unstable
           OH_SCAN_LN467MERGE:I.Data[5].2   // ISO/IEC15415 Unstable
           OH_SCAN_LN467MERGE:I.Data[5].3   // AIM DPM Unstable
           OH_SCAN_LN467MERGE:I.Data[5].4   // ADE AS9132 Unstable
           OH_SCAN_LN467MERGE:I.Data[5].5   // ISO/IEC15416 Unstable
           OH_SCAN_LN467MERGE:I.Data[5].6   // Reserved
           OH_SCAN_LN467MERGE:I.Data[5].7   // Reserved
           OH_SCAN_LN467MERGE:I.Data[6]   // Reserved
           OH_SCAN_LN467MERGE:I.Data[7]   // Reserved
           OH_SCAN_LN467MERGE:I.Data[8]   // Matching Level
           OH_SCAN_LN467MERGE:I.Data[9]   // Reserved
           OH_SCAN_LN467MERGE:O.Data[0].0   // Reserved
           OH_SCAN_LN467MERGE:O.Data[0].1   // Result Data Latch
           OH_SCAN_LN467MERGE:O.Data[0].2   // Reserved
           OH_SCAN_LN467MERGE:O.Data[0].3   // Reserved
           OH_SCAN_LN467MERGE:O.Data[0].4   // Reserved
           OH_SCAN_LN467MERGE:O.Data[0].5   // Reserved
           OH_SCAN_LN467MERGE:O.Data[0].6   // Reserved
           OH_SCAN_LN467MERGE:O.Data[0].7   // Error Clear
           OH_SCAN_LN467MERGE:O.Data[10]   // User Data Size
           OH_SCAN_LN467MERGE:O.Data[11]   // User Data Size
           OH_SCAN_LN467MERGE:O.Data[12]   // User Data
           OH_SCAN_LN467MERGE:O.Data[13]   // User Data
           OH_SCAN_LN467MERGE:O.Data[14]   // User Data
           OH_SCAN_LN467MERGE:O.Data[15]   // User Data
           OH_SCAN_LN467MERGE:O.Data[16]   // User Data
           OH_SCAN_LN467MERGE:O.Data[17]   // User Data
           OH_SCAN_LN467MERGE:O.Data[1].0   // Read Request
           OH_SCAN_LN467MERGE:O.Data[1].1   // Preset Request
           OH_SCAN_LN467MERGE:O.Data[1].2   // Register Preset Data Request
           OH_SCAN_LN467MERGE:O.Data[1].3   // Tune Request
           OH_SCAN_LN467MERGE:O.Data[1].4   // Bload Request
           OH_SCAN_LN467MERGE:O.Data[1].5   // Reserved
           OH_SCAN_LN467MERGE:O.Data[1].6   // Reserved
           OH_SCAN_LN467MERGE:O.Data[1].7   // Reserved
           OH_SCAN_LN467MERGE:O.Data[2].0   // Read Complete Clear
           OH_SCAN_LN467MERGE:O.Data[2].1   // Preset Complete Clear
           OH_SCAN_LN467MERGE:O.Data[2].2   // Register Preset Data Complete Clear
           OH_SCAN_LN467MERGE:O.Data[2].3   // Tune Complete Clear
           OH_SCAN_LN467MERGE:O.Data[2].4   // Bload Complete Clear
           OH_SCAN_LN467MERGE:O.Data[2].5   // Reserved
           OH_SCAN_LN467MERGE:O.Data[2].6   // Reserved
           OH_SCAN_LN467MERGE:O.Data[2].7   // External Request Complete Clear
           OH_SCAN_LN467MERGE:O.Data[3]   // Reserved
           OH_SCAN_LN467MERGE:O.Data[4]   // Bank Number
           OH_SCAN_LN467MERGE:O.Data[5]   // Bank Number
           OH_SCAN_LN467MERGE:O.Data[6]   // Reserved
           OH_SCAN_LN467MERGE:O.Data[7]   // Reserved
           OH_SCAN_LN467MERGE:O.Data[8]   // Reserved
           OH_SCAN_LN467MERGE:O.Data[9]   // Reserved
      OH_SCAN_LN7 : SR-2000 (Ethernet 10.28.160.140, rev 1.1, StandardDataDriven RPI 20 ms)
           OH_SCAN_LN7:I.Data[0].0   // Error
           OH_SCAN_LN7:I.Data[0].1   // Result Data Available
           OH_SCAN_LN7:I.Data[0].2   // Result Data Strobe
           OH_SCAN_LN7:I.Data[0].3   // Reserved
           OH_SCAN_LN7:I.Data[0].4   // Reserved
           OH_SCAN_LN7:I.Data[0].5   // Reserved
           OH_SCAN_LN7:I.Data[0].6   // Buffer Overflow Error
           OH_SCAN_LN7:I.Data[0].7   // General Error
           OH_SCAN_LN7:I.Data[10]   // ISO/IEC15415 Grade
           OH_SCAN_LN7:I.Data[11]   // Reserved
           OH_SCAN_LN7:I.Data[12]   // AIM DPM Grade
           OH_SCAN_LN7:I.Data[13]   // Reserved
           OH_SCAN_LN7:I.Data[14]   // ISO/IEC15416 Grade
           OH_SCAN_LN7:I.Data[15]   // Reserved
           OH_SCAN_LN7:I.Data[16]   // Read Result Code
           OH_SCAN_LN7:I.Data[17]   // Read Result Code
           OH_SCAN_LN7:I.Data[18]   // Preset Result Code
           OH_SCAN_LN7:I.Data[19]   // Preset Result Code
           OH_SCAN_LN7:I.Data[1].0   // Busy
           OH_SCAN_LN7:I.Data[1].1   // Trigger Busy
           OH_SCAN_LN7:I.Data[1].2   // Lock Busy
           OH_SCAN_LN7:I.Data[1].3   // Mode Busy
           OH_SCAN_LN7:I.Data[1].4   // Error Busy
           OH_SCAN_LN7:I.Data[1].5   // Reserved
           OH_SCAN_LN7:I.Data[1].6   // Ready
           OH_SCAN_LN7:I.Data[1].7   // Reserved
           OH_SCAN_LN7:I.Data[20]   // Register Preset Data Result Code
           OH_SCAN_LN7:I.Data[21]   // Register Preset Data Result Code
           OH_SCAN_LN7:I.Data[22]   // Tune Result Code
           OH_SCAN_LN7:I.Data[23]   // Tune Result Code
           OH_SCAN_LN7:I.Data[24]   // Bload Result Code
           OH_SCAN_LN7:I.Data[25]   // Bload Result Code
           OH_SCAN_LN7:I.Data[26]   // Reserved
           OH_SCAN_LN7:I.Data[27]   // Reserved
           OH_SCAN_LN7:I.Data[28]   // Reserved
           OH_SCAN_LN7:I.Data[29]   // Reserved
           OH_SCAN_LN7:I.Data[2].0   // Read Complete
           OH_SCAN_LN7:I.Data[2].1   // Preset Complete
           OH_SCAN_LN7:I.Data[2].2   // Register Preset Data Complete
           OH_SCAN_LN7:I.Data[2].3   // Tune Complete
           OH_SCAN_LN7:I.Data[2].4   // Bload Complete
           OH_SCAN_LN7:I.Data[2].5   // Reserved
           OH_SCAN_LN7:I.Data[2].6   // Reserved
           OH_SCAN_LN7:I.Data[2].7   // External Request Complete
           OH_SCAN_LN7:I.Data[30]   // External Request Result Code
           OH_SCAN_LN7:I.Data[31]   // External Request Result Code
           OH_SCAN_LN7:I.Data[32]   // General Error Code
           OH_SCAN_LN7:I.Data[33]   // General Error Code
           OH_SCAN_LN7:I.Data[34]   // Slave ID
           OH_SCAN_LN7:I.Data[35]   // Slave ID
           OH_SCAN_LN7:I.Data[36]   // Result Data Ready Count
           OH_SCAN_LN7:I.Data[37]   // Result Data Ready Count
           OH_SCAN_LN7:I.Data[38]   // Result Data Update Count
           OH_SCAN_LN7:I.Data[39]   // Result Data Update Count
           OH_SCAN_LN7:I.Data[3].0   // Read Failure
           OH_SCAN_LN7:I.Data[3].1   // Preset Failure
           OH_SCAN_LN7:I.Data[3].2   // Register Preset Data Failure
           OH_SCAN_LN7:I.Data[3].3   // Tune Failure
           OH_SCAN_LN7:I.Data[3].4   // Bload Failure
           OH_SCAN_LN7:I.Data[3].5   // Reserved
           OH_SCAN_LN7:I.Data[3].6   // Reserved
           OH_SCAN_LN7:I.Data[3].7   // External Request Failure
           OH_SCAN_LN7:I.Data[40]   // Trigger Input Count for Master
           OH_SCAN_LN7:I.Data[41]   // Trigger Input Count for Master
           OH_SCAN_LN7:I.Data[42]   // Result Data Size
           OH_SCAN_LN7:I.Data[43]   // Result Data Size
           OH_SCAN_LN7:I.Data[44]   // Result Data
           OH_SCAN_LN7:I.Data[45]   // Result Data
           OH_SCAN_LN7:I.Data[46]   // Result Data
           OH_SCAN_LN7:I.Data[47]   // Result Data
           OH_SCAN_LN7:I.Data[48]   // Result Data
           OH_SCAN_LN7:I.Data[49]   // Result Data
           OH_SCAN_LN7:I.Data[4].0   // Input 1 Status
           OH_SCAN_LN7:I.Data[4].1   // Input 2 Status
           OH_SCAN_LN7:I.Data[4].2   // Reserved
           OH_SCAN_LN7:I.Data[4].3   // Reserved
           OH_SCAN_LN7:I.Data[4].4   // Output 1 Status
           OH_SCAN_LN7:I.Data[4].5   // Output 2 Status
           OH_SCAN_LN7:I.Data[4].6   // Output 3 Status
           OH_SCAN_LN7:I.Data[4].7   // Reserved
           OH_SCAN_LN7:I.Data[50]   // Result Data
           OH_SCAN_LN7:I.Data[5].0   // Unstable
           OH_SCAN_LN7:I.Data[5].1   // Matching Level Unstable
           OH_SCAN_LN7:I.Data[5].2   // ISO/IEC15415 Unstable
           OH_SCAN_LN7:I.Data[5].3   // AIM DPM Unstable
           OH_SCAN_LN7:I.Data[5].4   // ADE AS9132 Unstable
           OH_SCAN_LN7:I.Data[5].5   // ISO/IEC15416 Unstable
           OH_SCAN_LN7:I.Data[5].6   // Reserved
           OH_SCAN_LN7:I.Data[5].7   // Reserved
           OH_SCAN_LN7:I.Data[6]   // Reserved
           OH_SCAN_LN7:I.Data[7]   // Reserved
           OH_SCAN_LN7:I.Data[8]   // Matching Level
           OH_SCAN_LN7:I.Data[9]   // Reserved
           OH_SCAN_LN7:O.Data[0].0   // Reserved
           OH_SCAN_LN7:O.Data[0].1   // Result Data Latch
           OH_SCAN_LN7:O.Data[0].2   // Reserved
           OH_SCAN_LN7:O.Data[0].3   // Reserved
           OH_SCAN_LN7:O.Data[0].4   // Reserved
           OH_SCAN_LN7:O.Data[0].5   // Reserved
           OH_SCAN_LN7:O.Data[0].6   // Reserved
           OH_SCAN_LN7:O.Data[0].7   // Error Clear
           OH_SCAN_LN7:O.Data[10]   // User Data Size
           OH_SCAN_LN7:O.Data[11]   // User Data Size
           OH_SCAN_LN7:O.Data[12]   // User Data
           OH_SCAN_LN7:O.Data[13]   // User Data
           OH_SCAN_LN7:O.Data[14]   // User Data
           OH_SCAN_LN7:O.Data[15]   // User Data
           OH_SCAN_LN7:O.Data[16]   // User Data
           OH_SCAN_LN7:O.Data[17]   // User Data
           OH_SCAN_LN7:O.Data[1].0   // Read Request
           OH_SCAN_LN7:O.Data[1].1   // Preset Request
           OH_SCAN_LN7:O.Data[1].2   // Register Preset Data Request
           OH_SCAN_LN7:O.Data[1].3   // Tune Request
           OH_SCAN_LN7:O.Data[1].4   // Bload Request
           OH_SCAN_LN7:O.Data[1].5   // Reserved
           OH_SCAN_LN7:O.Data[1].6   // Reserved
           OH_SCAN_LN7:O.Data[1].7   // Reserved
           OH_SCAN_LN7:O.Data[2].0   // Read Complete Clear
           OH_SCAN_LN7:O.Data[2].1   // Preset Complete Clear
           OH_SCAN_LN7:O.Data[2].2   // Register Preset Data Complete Clear
           OH_SCAN_LN7:O.Data[2].3   // Tune Complete Clear
           OH_SCAN_LN7:O.Data[2].4   // Bload Complete Clear
           OH_SCAN_LN7:O.Data[2].5   // Reserved
           OH_SCAN_LN7:O.Data[2].6   // Reserved
           OH_SCAN_LN7:O.Data[2].7   // External Request Complete Clear
           OH_SCAN_LN7:O.Data[3]   // Reserved
           OH_SCAN_LN7:O.Data[4]   // Bank Number
           OH_SCAN_LN7:O.Data[5]   // Bank Number
           OH_SCAN_LN7:O.Data[6]   // Reserved
           OH_SCAN_LN7:O.Data[7]   // Reserved
           OH_SCAN_LN7:O.Data[8]   // Reserved
           OH_SCAN_LN7:O.Data[9]   // Reserved
      OH_SCAN_CLEARPACK : SR-2000 (Ethernet 10.28.17.143, rev 1.1, StandardDataDriven RPI 20 ms)
           OH_SCAN_CLEARPACK:I.Data[0].0   // Error
           OH_SCAN_CLEARPACK:I.Data[0].1   // Result Data Available
           OH_SCAN_CLEARPACK:I.Data[0].2   // Result Data Strobe
           OH_SCAN_CLEARPACK:I.Data[0].3   // Reserved
           OH_SCAN_CLEARPACK:I.Data[0].4   // Reserved
           OH_SCAN_CLEARPACK:I.Data[0].5   // Reserved
           OH_SCAN_CLEARPACK:I.Data[0].6   // Buffer Overflow Error
           OH_SCAN_CLEARPACK:I.Data[0].7   // General Error
           OH_SCAN_CLEARPACK:I.Data[10]   // ISO/IEC15415 Grade
           OH_SCAN_CLEARPACK:I.Data[11]   // Reserved
           OH_SCAN_CLEARPACK:I.Data[12]   // AIM DPM Grade
           OH_SCAN_CLEARPACK:I.Data[13]   // Reserved
           OH_SCAN_CLEARPACK:I.Data[14]   // ISO/IEC15416 Grade
           OH_SCAN_CLEARPACK:I.Data[15]   // Reserved
           OH_SCAN_CLEARPACK:I.Data[16]   // Read Result Code
           OH_SCAN_CLEARPACK:I.Data[17]   // Read Result Code
           OH_SCAN_CLEARPACK:I.Data[18]   // Preset Result Code
           OH_SCAN_CLEARPACK:I.Data[19]   // Preset Result Code
           OH_SCAN_CLEARPACK:I.Data[1].0   // Busy
           OH_SCAN_CLEARPACK:I.Data[1].1   // Trigger Busy
           OH_SCAN_CLEARPACK:I.Data[1].2   // Lock Busy
           OH_SCAN_CLEARPACK:I.Data[1].3   // Mode Busy
           OH_SCAN_CLEARPACK:I.Data[1].4   // Error Busy
           OH_SCAN_CLEARPACK:I.Data[1].5   // Reserved
           OH_SCAN_CLEARPACK:I.Data[1].6   // Ready
           OH_SCAN_CLEARPACK:I.Data[1].7   // Reserved
           OH_SCAN_CLEARPACK:I.Data[20]   // Register Preset Data Result Code
           OH_SCAN_CLEARPACK:I.Data[21]   // Register Preset Data Result Code
           OH_SCAN_CLEARPACK:I.Data[22]   // Tune Result Code
           OH_SCAN_CLEARPACK:I.Data[23]   // Tune Result Code
           OH_SCAN_CLEARPACK:I.Data[24]   // Bload Result Code
           OH_SCAN_CLEARPACK:I.Data[25]   // Bload Result Code
           OH_SCAN_CLEARPACK:I.Data[26]   // Reserved
           OH_SCAN_CLEARPACK:I.Data[27]   // Reserved
           OH_SCAN_CLEARPACK:I.Data[28]   // Reserved
           OH_SCAN_CLEARPACK:I.Data[29]   // Reserved
           OH_SCAN_CLEARPACK:I.Data[2].0   // Read Complete
           OH_SCAN_CLEARPACK:I.Data[2].1   // Preset Complete
           OH_SCAN_CLEARPACK:I.Data[2].2   // Register Preset Data Complete
           OH_SCAN_CLEARPACK:I.Data[2].3   // Tune Complete
           OH_SCAN_CLEARPACK:I.Data[2].4   // Bload Complete
           OH_SCAN_CLEARPACK:I.Data[2].5   // Reserved
           OH_SCAN_CLEARPACK:I.Data[2].6   // Reserved
           OH_SCAN_CLEARPACK:I.Data[2].7   // External Request Complete
           OH_SCAN_CLEARPACK:I.Data[30]   // External Request Result Code
           OH_SCAN_CLEARPACK:I.Data[31]   // External Request Result Code
           OH_SCAN_CLEARPACK:I.Data[32]   // General Error Code
           OH_SCAN_CLEARPACK:I.Data[33]   // General Error Code
           OH_SCAN_CLEARPACK:I.Data[34]   // Slave ID
           OH_SCAN_CLEARPACK:I.Data[35]   // Slave ID
           OH_SCAN_CLEARPACK:I.Data[36]   // Result Data Ready Count
           OH_SCAN_CLEARPACK:I.Data[37]   // Result Data Ready Count
           OH_SCAN_CLEARPACK:I.Data[38]   // Result Data Update Count
           OH_SCAN_CLEARPACK:I.Data[39]   // Result Data Update Count
           OH_SCAN_CLEARPACK:I.Data[3].0   // Read Failure
           OH_SCAN_CLEARPACK:I.Data[3].1   // Preset Failure
           OH_SCAN_CLEARPACK:I.Data[3].2   // Register Preset Data Failure
           OH_SCAN_CLEARPACK:I.Data[3].3   // Tune Failure
           OH_SCAN_CLEARPACK:I.Data[3].4   // Bload Failure
           OH_SCAN_CLEARPACK:I.Data[3].5   // Reserved
           OH_SCAN_CLEARPACK:I.Data[3].6   // Reserved
           OH_SCAN_CLEARPACK:I.Data[3].7   // External Request Failure
           OH_SCAN_CLEARPACK:I.Data[40]   // Trigger Input Count for Master
           OH_SCAN_CLEARPACK:I.Data[41]   // Trigger Input Count for Master
           OH_SCAN_CLEARPACK:I.Data[42]   // Result Data Size
           OH_SCAN_CLEARPACK:I.Data[43]   // Result Data Size
           OH_SCAN_CLEARPACK:I.Data[44]   // Result Data
           OH_SCAN_CLEARPACK:I.Data[45]   // Result Data
           OH_SCAN_CLEARPACK:I.Data[46]   // Result Data
           OH_SCAN_CLEARPACK:I.Data[47]   // Result Data
           OH_SCAN_CLEARPACK:I.Data[48]   // Result Data
           OH_SCAN_CLEARPACK:I.Data[49]   // Result Data
           OH_SCAN_CLEARPACK:I.Data[4].0   // Input 1 Status
           OH_SCAN_CLEARPACK:I.Data[4].1   // Input 2 Status
           OH_SCAN_CLEARPACK:I.Data[4].2   // Reserved
           OH_SCAN_CLEARPACK:I.Data[4].3   // Reserved
           OH_SCAN_CLEARPACK:I.Data[4].4   // Output 1 Status
           OH_SCAN_CLEARPACK:I.Data[4].5   // Output 2 Status
           OH_SCAN_CLEARPACK:I.Data[4].6   // Output 3 Status
           OH_SCAN_CLEARPACK:I.Data[4].7   // Reserved
           OH_SCAN_CLEARPACK:I.Data[50]   // Result Data
           OH_SCAN_CLEARPACK:I.Data[5].0   // Unstable
           OH_SCAN_CLEARPACK:I.Data[5].1   // Matching Level Unstable
           OH_SCAN_CLEARPACK:I.Data[5].2   // ISO/IEC15415 Unstable
           OH_SCAN_CLEARPACK:I.Data[5].3   // AIM DPM Unstable
           OH_SCAN_CLEARPACK:I.Data[5].4   // ADE AS9132 Unstable
           OH_SCAN_CLEARPACK:I.Data[5].5   // ISO/IEC15416 Unstable
           OH_SCAN_CLEARPACK:I.Data[5].6   // Reserved
           OH_SCAN_CLEARPACK:I.Data[5].7   // Reserved
           OH_SCAN_CLEARPACK:I.Data[6]   // Reserved
           OH_SCAN_CLEARPACK:I.Data[7]   // Reserved
           OH_SCAN_CLEARPACK:I.Data[8]   // Matching Level
           OH_SCAN_CLEARPACK:I.Data[9]   // Reserved
           OH_SCAN_CLEARPACK:O.Data[0].0   // Reserved
           OH_SCAN_CLEARPACK:O.Data[0].1   // Result Data Latch
           OH_SCAN_CLEARPACK:O.Data[0].2   // Reserved
           OH_SCAN_CLEARPACK:O.Data[0].3   // Reserved
           OH_SCAN_CLEARPACK:O.Data[0].4   // Reserved
           OH_SCAN_CLEARPACK:O.Data[0].5   // Reserved
           OH_SCAN_CLEARPACK:O.Data[0].6   // Reserved
           OH_SCAN_CLEARPACK:O.Data[0].7   // Error Clear
           OH_SCAN_CLEARPACK:O.Data[10]   // User Data Size
           OH_SCAN_CLEARPACK:O.Data[11]   // User Data Size
           OH_SCAN_CLEARPACK:O.Data[12]   // User Data
           OH_SCAN_CLEARPACK:O.Data[13]   // User Data
           OH_SCAN_CLEARPACK:O.Data[14]   // User Data
           OH_SCAN_CLEARPACK:O.Data[15]   // User Data
           OH_SCAN_CLEARPACK:O.Data[16]   // User Data
           OH_SCAN_CLEARPACK:O.Data[17]   // User Data
           OH_SCAN_CLEARPACK:O.Data[1].0   // Read Request
           OH_SCAN_CLEARPACK:O.Data[1].1   // Preset Request
           OH_SCAN_CLEARPACK:O.Data[1].2   // Register Preset Data Request
           OH_SCAN_CLEARPACK:O.Data[1].3   // Tune Request
           OH_SCAN_CLEARPACK:O.Data[1].4   // Bload Request
           OH_SCAN_CLEARPACK:O.Data[1].5   // Reserved
           OH_SCAN_CLEARPACK:O.Data[1].6   // Reserved
           OH_SCAN_CLEARPACK:O.Data[1].7   // Reserved
           OH_SCAN_CLEARPACK:O.Data[2].0   // Read Complete Clear
           OH_SCAN_CLEARPACK:O.Data[2].1   // Preset Complete Clear
           OH_SCAN_CLEARPACK:O.Data[2].2   // Register Preset Data Complete Clear
           OH_SCAN_CLEARPACK:O.Data[2].3   // Tune Complete Clear
           OH_SCAN_CLEARPACK:O.Data[2].4   // Bload Complete Clear
           OH_SCAN_CLEARPACK:O.Data[2].5   // Reserved
           OH_SCAN_CLEARPACK:O.Data[2].6   // Reserved
           OH_SCAN_CLEARPACK:O.Data[2].7   // External Request Complete Clear
           OH_SCAN_CLEARPACK:O.Data[3]   // Reserved
           OH_SCAN_CLEARPACK:O.Data[4]   // Bank Number
           OH_SCAN_CLEARPACK:O.Data[5]   // Bank Number
           OH_SCAN_CLEARPACK:O.Data[6]   // Reserved
           OH_SCAN_CLEARPACK:O.Data[7]   // Reserved
           OH_SCAN_CLEARPACK:O.Data[8]   // Reserved
           OH_SCAN_CLEARPACK:O.Data[9]   // Reserved
      OH_SCAN_LONGTERMWEST : SR-2000 (Ethernet 10.28.17.141, rev 1.1, StandardDataDriven RPI 20 ms)
           OH_SCAN_LONGTERMWEST:I.Data[0].0   // Error
           OH_SCAN_LONGTERMWEST:I.Data[0].1   // Result Data Available
           OH_SCAN_LONGTERMWEST:I.Data[0].2   // Result Data Strobe
           OH_SCAN_LONGTERMWEST:I.Data[0].3   // Reserved
           OH_SCAN_LONGTERMWEST:I.Data[0].4   // Reserved
           OH_SCAN_LONGTERMWEST:I.Data[0].5   // Reserved
           OH_SCAN_LONGTERMWEST:I.Data[0].6   // Buffer Overflow Error
           OH_SCAN_LONGTERMWEST:I.Data[0].7   // General Error
           OH_SCAN_LONGTERMWEST:I.Data[10]   // ISO/IEC15415 Grade
           OH_SCAN_LONGTERMWEST:I.Data[11]   // Reserved
           OH_SCAN_LONGTERMWEST:I.Data[12]   // AIM DPM Grade
           OH_SCAN_LONGTERMWEST:I.Data[13]   // Reserved
           OH_SCAN_LONGTERMWEST:I.Data[14]   // ISO/IEC15416 Grade
           OH_SCAN_LONGTERMWEST:I.Data[15]   // Reserved
           OH_SCAN_LONGTERMWEST:I.Data[16]   // Read Result Code
           OH_SCAN_LONGTERMWEST:I.Data[17]   // Read Result Code
           OH_SCAN_LONGTERMWEST:I.Data[18]   // Preset Result Code
           OH_SCAN_LONGTERMWEST:I.Data[19]   // Preset Result Code
           OH_SCAN_LONGTERMWEST:I.Data[1].0   // Busy
           OH_SCAN_LONGTERMWEST:I.Data[1].1   // Trigger Busy
           OH_SCAN_LONGTERMWEST:I.Data[1].2   // Lock Busy
           OH_SCAN_LONGTERMWEST:I.Data[1].3   // Mode Busy
           OH_SCAN_LONGTERMWEST:I.Data[1].4   // Error Busy
           OH_SCAN_LONGTERMWEST:I.Data[1].5   // Reserved
           OH_SCAN_LONGTERMWEST:I.Data[1].6   // Ready
           OH_SCAN_LONGTERMWEST:I.Data[1].7   // Reserved
           OH_SCAN_LONGTERMWEST:I.Data[20]   // Register Preset Data Result Code
           OH_SCAN_LONGTERMWEST:I.Data[21]   // Register Preset Data Result Code
           OH_SCAN_LONGTERMWEST:I.Data[22]   // Tune Result Code
           OH_SCAN_LONGTERMWEST:I.Data[23]   // Tune Result Code
           OH_SCAN_LONGTERMWEST:I.Data[24]   // Bload Result Code
           OH_SCAN_LONGTERMWEST:I.Data[25]   // Bload Result Code
           OH_SCAN_LONGTERMWEST:I.Data[26]   // Reserved
           OH_SCAN_LONGTERMWEST:I.Data[27]   // Reserved
           OH_SCAN_LONGTERMWEST:I.Data[28]   // Reserved
           OH_SCAN_LONGTERMWEST:I.Data[29]   // Reserved
           OH_SCAN_LONGTERMWEST:I.Data[2].0   // Read Complete
           OH_SCAN_LONGTERMWEST:I.Data[2].1   // Preset Complete
           OH_SCAN_LONGTERMWEST:I.Data[2].2   // Register Preset Data Complete
           OH_SCAN_LONGTERMWEST:I.Data[2].3   // Tune Complete
           OH_SCAN_LONGTERMWEST:I.Data[2].4   // Bload Complete
           OH_SCAN_LONGTERMWEST:I.Data[2].5   // Reserved
           OH_SCAN_LONGTERMWEST:I.Data[2].6   // Reserved
           OH_SCAN_LONGTERMWEST:I.Data[2].7   // External Request Complete
           OH_SCAN_LONGTERMWEST:I.Data[30]   // External Request Result Code
           OH_SCAN_LONGTERMWEST:I.Data[31]   // External Request Result Code
           OH_SCAN_LONGTERMWEST:I.Data[32]   // General Error Code
           OH_SCAN_LONGTERMWEST:I.Data[33]   // General Error Code
           OH_SCAN_LONGTERMWEST:I.Data[34]   // Slave ID
           OH_SCAN_LONGTERMWEST:I.Data[35]   // Slave ID
           OH_SCAN_LONGTERMWEST:I.Data[36]   // Result Data Ready Count
           OH_SCAN_LONGTERMWEST:I.Data[37]   // Result Data Ready Count
           OH_SCAN_LONGTERMWEST:I.Data[38]   // Result Data Update Count
           OH_SCAN_LONGTERMWEST:I.Data[39]   // Result Data Update Count
           OH_SCAN_LONGTERMWEST:I.Data[3].0   // Read Failure
           OH_SCAN_LONGTERMWEST:I.Data[3].1   // Preset Failure
           OH_SCAN_LONGTERMWEST:I.Data[3].2   // Register Preset Data Failure
           OH_SCAN_LONGTERMWEST:I.Data[3].3   // Tune Failure
           OH_SCAN_LONGTERMWEST:I.Data[3].4   // Bload Failure
           OH_SCAN_LONGTERMWEST:I.Data[3].5   // Reserved
           OH_SCAN_LONGTERMWEST:I.Data[3].6   // Reserved
           OH_SCAN_LONGTERMWEST:I.Data[3].7   // External Request Failure
           OH_SCAN_LONGTERMWEST:I.Data[40]   // Trigger Input Count for Master
           OH_SCAN_LONGTERMWEST:I.Data[41]   // Trigger Input Count for Master
           OH_SCAN_LONGTERMWEST:I.Data[42]   // Result Data Size
           OH_SCAN_LONGTERMWEST:I.Data[43]   // Result Data Size
           OH_SCAN_LONGTERMWEST:I.Data[44]   // Result Data
           OH_SCAN_LONGTERMWEST:I.Data[45]   // Result Data
           OH_SCAN_LONGTERMWEST:I.Data[46]   // Result Data
           OH_SCAN_LONGTERMWEST:I.Data[47]   // Result Data
           OH_SCAN_LONGTERMWEST:I.Data[48]   // Result Data
           OH_SCAN_LONGTERMWEST:I.Data[49]   // Result Data
           OH_SCAN_LONGTERMWEST:I.Data[4].0   // Input 1 Status
           OH_SCAN_LONGTERMWEST:I.Data[4].1   // Input 2 Status
           OH_SCAN_LONGTERMWEST:I.Data[4].2   // Reserved
           OH_SCAN_LONGTERMWEST:I.Data[4].3   // Reserved
           OH_SCAN_LONGTERMWEST:I.Data[4].4   // Output 1 Status
           OH_SCAN_LONGTERMWEST:I.Data[4].5   // Output 2 Status
           OH_SCAN_LONGTERMWEST:I.Data[4].6   // Output 3 Status
           OH_SCAN_LONGTERMWEST:I.Data[4].7   // Reserved
           OH_SCAN_LONGTERMWEST:I.Data[50]   // Result Data
           OH_SCAN_LONGTERMWEST:I.Data[5].0   // Unstable
           OH_SCAN_LONGTERMWEST:I.Data[5].1   // Matching Level Unstable
           OH_SCAN_LONGTERMWEST:I.Data[5].2   // ISO/IEC15415 Unstable
           OH_SCAN_LONGTERMWEST:I.Data[5].3   // AIM DPM Unstable
           OH_SCAN_LONGTERMWEST:I.Data[5].4   // ADE AS9132 Unstable
           OH_SCAN_LONGTERMWEST:I.Data[5].5   // ISO/IEC15416 Unstable
           OH_SCAN_LONGTERMWEST:I.Data[5].6   // Reserved
           OH_SCAN_LONGTERMWEST:I.Data[5].7   // Reserved
           OH_SCAN_LONGTERMWEST:I.Data[6]   // Reserved
           OH_SCAN_LONGTERMWEST:I.Data[7]   // Reserved
           OH_SCAN_LONGTERMWEST:I.Data[8]   // Matching Level
           OH_SCAN_LONGTERMWEST:I.Data[9]   // Reserved
           OH_SCAN_LONGTERMWEST:O.Data[0].0   // Reserved
           OH_SCAN_LONGTERMWEST:O.Data[0].1   // Result Data Latch
           OH_SCAN_LONGTERMWEST:O.Data[0].2   // Reserved
           OH_SCAN_LONGTERMWEST:O.Data[0].3   // Reserved
           OH_SCAN_LONGTERMWEST:O.Data[0].4   // Reserved
           OH_SCAN_LONGTERMWEST:O.Data[0].5   // Reserved
           OH_SCAN_LONGTERMWEST:O.Data[0].6   // Reserved
           OH_SCAN_LONGTERMWEST:O.Data[0].7   // Error Clear
           OH_SCAN_LONGTERMWEST:O.Data[10]   // User Data Size
           OH_SCAN_LONGTERMWEST:O.Data[11]   // User Data Size
           OH_SCAN_LONGTERMWEST:O.Data[12]   // User Data
           OH_SCAN_LONGTERMWEST:O.Data[13]   // User Data
           OH_SCAN_LONGTERMWEST:O.Data[14]   // User Data
           OH_SCAN_LONGTERMWEST:O.Data[15]   // User Data
           OH_SCAN_LONGTERMWEST:O.Data[16]   // User Data
           OH_SCAN_LONGTERMWEST:O.Data[17]   // User Data
           OH_SCAN_LONGTERMWEST:O.Data[1].0   // Read Request
           OH_SCAN_LONGTERMWEST:O.Data[1].1   // Preset Request
           OH_SCAN_LONGTERMWEST:O.Data[1].2   // Register Preset Data Request
           OH_SCAN_LONGTERMWEST:O.Data[1].3   // Tune Request
           OH_SCAN_LONGTERMWEST:O.Data[1].4   // Bload Request
           OH_SCAN_LONGTERMWEST:O.Data[1].5   // Reserved
           OH_SCAN_LONGTERMWEST:O.Data[1].6   // Reserved
           OH_SCAN_LONGTERMWEST:O.Data[1].7   // Reserved
           OH_SCAN_LONGTERMWEST:O.Data[2].0   // Read Complete Clear
           OH_SCAN_LONGTERMWEST:O.Data[2].1   // Preset Complete Clear
           OH_SCAN_LONGTERMWEST:O.Data[2].2   // Register Preset Data Complete Clear
           OH_SCAN_LONGTERMWEST:O.Data[2].3   // Tune Complete Clear
           OH_SCAN_LONGTERMWEST:O.Data[2].4   // Bload Complete Clear
           OH_SCAN_LONGTERMWEST:O.Data[2].5   // Reserved
           OH_SCAN_LONGTERMWEST:O.Data[2].6   // Reserved
           OH_SCAN_LONGTERMWEST:O.Data[2].7   // External Request Complete Clear
           OH_SCAN_LONGTERMWEST:O.Data[3]   // Reserved
           OH_SCAN_LONGTERMWEST:O.Data[4]   // Bank Number
           OH_SCAN_LONGTERMWEST:O.Data[5]   // Bank Number
           OH_SCAN_LONGTERMWEST:O.Data[6]   // Reserved
           OH_SCAN_LONGTERMWEST:O.Data[7]   // Reserved
           OH_SCAN_LONGTERMWEST:O.Data[8]   // Reserved
           OH_SCAN_LONGTERMWEST:O.Data[9]   // Reserved
      OH_SCAN_LN4 : SR-2000 (Ethernet 10.28.88.201, rev 1.1, StandardDataDriven RPI 20 ms)
           OH_SCAN_LN4:I.Data[0].0   // Error
           OH_SCAN_LN4:I.Data[0].1   // Result Data Available
           OH_SCAN_LN4:I.Data[0].2   // Result Data Strobe
           OH_SCAN_LN4:I.Data[0].3   // Reserved
           OH_SCAN_LN4:I.Data[0].4   // Reserved
           OH_SCAN_LN4:I.Data[0].5   // Reserved
           OH_SCAN_LN4:I.Data[0].6   // Buffer Overflow Error
           OH_SCAN_LN4:I.Data[0].7   // General Error
           OH_SCAN_LN4:I.Data[10]   // ISO/IEC15415 Grade
           OH_SCAN_LN4:I.Data[11]   // Reserved
           OH_SCAN_LN4:I.Data[12]   // AIM DPM Grade
           OH_SCAN_LN4:I.Data[13]   // Reserved
           OH_SCAN_LN4:I.Data[14]   // ISO/IEC15416 Grade
           OH_SCAN_LN4:I.Data[15]   // Reserved
           OH_SCAN_LN4:I.Data[16]   // Read Result Code
           OH_SCAN_LN4:I.Data[17]   // Read Result Code
           OH_SCAN_LN4:I.Data[18]   // Preset Result Code
           OH_SCAN_LN4:I.Data[19]   // Preset Result Code
           OH_SCAN_LN4:I.Data[1].0   // Busy
           OH_SCAN_LN4:I.Data[1].1   // Trigger Busy
           OH_SCAN_LN4:I.Data[1].2   // Lock Busy
           OH_SCAN_LN4:I.Data[1].3   // Mode Busy
           OH_SCAN_LN4:I.Data[1].4   // Error Busy
           OH_SCAN_LN4:I.Data[1].5   // Reserved
           OH_SCAN_LN4:I.Data[1].6   // Ready
           OH_SCAN_LN4:I.Data[1].7   // Reserved
           OH_SCAN_LN4:I.Data[20]   // Register Preset Data Result Code
           OH_SCAN_LN4:I.Data[21]   // Register Preset Data Result Code
           OH_SCAN_LN4:I.Data[22]   // Tune Result Code
           OH_SCAN_LN4:I.Data[23]   // Tune Result Code
           OH_SCAN_LN4:I.Data[24]   // Bload Result Code
           OH_SCAN_LN4:I.Data[25]   // Bload Result Code
           OH_SCAN_LN4:I.Data[26]   // Reserved
           OH_SCAN_LN4:I.Data[27]   // Reserved
           OH_SCAN_LN4:I.Data[28]   // Reserved
           OH_SCAN_LN4:I.Data[29]   // Reserved
           OH_SCAN_LN4:I.Data[2].0   // Read Complete
           OH_SCAN_LN4:I.Data[2].1   // Preset Complete
           OH_SCAN_LN4:I.Data[2].2   // Register Preset Data Complete
           OH_SCAN_LN4:I.Data[2].3   // Tune Complete
           OH_SCAN_LN4:I.Data[2].4   // Bload Complete
           OH_SCAN_LN4:I.Data[2].5   // Reserved
           OH_SCAN_LN4:I.Data[2].6   // Reserved
           OH_SCAN_LN4:I.Data[2].7   // External Request Complete
           OH_SCAN_LN4:I.Data[30]   // External Request Result Code
           OH_SCAN_LN4:I.Data[31]   // External Request Result Code
           OH_SCAN_LN4:I.Data[32]   // General Error Code
           OH_SCAN_LN4:I.Data[33]   // General Error Code
           OH_SCAN_LN4:I.Data[34]   // Slave ID
           OH_SCAN_LN4:I.Data[35]   // Slave ID
           OH_SCAN_LN4:I.Data[36]   // Result Data Ready Count
           OH_SCAN_LN4:I.Data[37]   // Result Data Ready Count
           OH_SCAN_LN4:I.Data[38]   // Result Data Update Count
           OH_SCAN_LN4:I.Data[39]   // Result Data Update Count
           OH_SCAN_LN4:I.Data[3].0   // Read Failure
           OH_SCAN_LN4:I.Data[3].1   // Preset Failure
           OH_SCAN_LN4:I.Data[3].2   // Register Preset Data Failure
           OH_SCAN_LN4:I.Data[3].3   // Tune Failure
           OH_SCAN_LN4:I.Data[3].4   // Bload Failure
           OH_SCAN_LN4:I.Data[3].5   // Reserved
           OH_SCAN_LN4:I.Data[3].6   // Reserved
           OH_SCAN_LN4:I.Data[3].7   // External Request Failure
           OH_SCAN_LN4:I.Data[40]   // Trigger Input Count for Master
           OH_SCAN_LN4:I.Data[41]   // Trigger Input Count for Master
           OH_SCAN_LN4:I.Data[42]   // Result Data Size
           OH_SCAN_LN4:I.Data[43]   // Result Data Size
           OH_SCAN_LN4:I.Data[44]   // Result Data
           OH_SCAN_LN4:I.Data[45]   // Result Data
           OH_SCAN_LN4:I.Data[46]   // Result Data
           OH_SCAN_LN4:I.Data[47]   // Result Data
           OH_SCAN_LN4:I.Data[48]   // Result Data
           OH_SCAN_LN4:I.Data[49]   // Result Data
           OH_SCAN_LN4:I.Data[4].0   // Input 1 Status
           OH_SCAN_LN4:I.Data[4].1   // Input 2 Status
           OH_SCAN_LN4:I.Data[4].2   // Reserved
           OH_SCAN_LN4:I.Data[4].3   // Reserved
           OH_SCAN_LN4:I.Data[4].4   // Output 1 Status
           OH_SCAN_LN4:I.Data[4].5   // Output 2 Status
           OH_SCAN_LN4:I.Data[4].6   // Output 3 Status
           OH_SCAN_LN4:I.Data[4].7   // Reserved
           OH_SCAN_LN4:I.Data[50]   // Result Data
           OH_SCAN_LN4:I.Data[5].0   // Unstable
           OH_SCAN_LN4:I.Data[5].1   // Matching Level Unstable
           OH_SCAN_LN4:I.Data[5].2   // ISO/IEC15415 Unstable
           OH_SCAN_LN4:I.Data[5].3   // AIM DPM Unstable
           OH_SCAN_LN4:I.Data[5].4   // ADE AS9132 Unstable
           OH_SCAN_LN4:I.Data[5].5   // ISO/IEC15416 Unstable
           OH_SCAN_LN4:I.Data[5].6   // Reserved
           OH_SCAN_LN4:I.Data[5].7   // Reserved
           OH_SCAN_LN4:I.Data[6]   // Reserved
           OH_SCAN_LN4:I.Data[7]   // Reserved
           OH_SCAN_LN4:I.Data[8]   // Matching Level
           OH_SCAN_LN4:I.Data[9]   // Reserved
           OH_SCAN_LN4:O.Data[0].0   // Reserved
           OH_SCAN_LN4:O.Data[0].1   // Result Data Latch
           OH_SCAN_LN4:O.Data[0].2   // Reserved
           OH_SCAN_LN4:O.Data[0].3   // Reserved
           OH_SCAN_LN4:O.Data[0].4   // Reserved
           OH_SCAN_LN4:O.Data[0].5   // Reserved
           OH_SCAN_LN4:O.Data[0].6   // Reserved
           OH_SCAN_LN4:O.Data[0].7   // Error Clear
           OH_SCAN_LN4:O.Data[10]   // User Data Size
           OH_SCAN_LN4:O.Data[11]   // User Data Size
           OH_SCAN_LN4:O.Data[12]   // User Data
           OH_SCAN_LN4:O.Data[13]   // User Data
           OH_SCAN_LN4:O.Data[14]   // User Data
           OH_SCAN_LN4:O.Data[15]   // User Data
           OH_SCAN_LN4:O.Data[16]   // User Data
           OH_SCAN_LN4:O.Data[17]   // User Data
           OH_SCAN_LN4:O.Data[1].0   // Read Request
           OH_SCAN_LN4:O.Data[1].1   // Preset Request
           OH_SCAN_LN4:O.Data[1].2   // Register Preset Data Request
           OH_SCAN_LN4:O.Data[1].3   // Tune Request
           OH_SCAN_LN4:O.Data[1].4   // Bload Request
           OH_SCAN_LN4:O.Data[1].5   // Reserved
           OH_SCAN_LN4:O.Data[1].6   // Reserved
           OH_SCAN_LN4:O.Data[1].7   // Reserved
           OH_SCAN_LN4:O.Data[2].0   // Read Complete Clear
           OH_SCAN_LN4:O.Data[2].1   // Preset Complete Clear
           OH_SCAN_LN4:O.Data[2].2   // Register Preset Data Complete Clear
           OH_SCAN_LN4:O.Data[2].3   // Tune Complete Clear
           OH_SCAN_LN4:O.Data[2].4   // Bload Complete Clear
           OH_SCAN_LN4:O.Data[2].5   // Reserved
           OH_SCAN_LN4:O.Data[2].6   // Reserved
           OH_SCAN_LN4:O.Data[2].7   // External Request Complete Clear
           OH_SCAN_LN4:O.Data[3]   // Reserved
           OH_SCAN_LN4:O.Data[4]   // Bank Number
           OH_SCAN_LN4:O.Data[5]   // Bank Number
           OH_SCAN_LN4:O.Data[6]   // Reserved
           OH_SCAN_LN4:O.Data[7]   // Reserved
           OH_SCAN_LN4:O.Data[8]   // Reserved
           OH_SCAN_LN4:O.Data[9]   // Reserved
      OH_SCAN_WAREHOUSESOUTH : SR-2000 (Ethernet 10.28.17.139, rev 1.1, StandardDataDriven RPI 20 ms)
           OH_SCAN_WAREHOUSESOUTH:I.Data[0].0   // Error
           OH_SCAN_WAREHOUSESOUTH:I.Data[0].1   // Result Data Available
           OH_SCAN_WAREHOUSESOUTH:I.Data[0].2   // Result Data Strobe
           OH_SCAN_WAREHOUSESOUTH:I.Data[0].3   // Reserved
           OH_SCAN_WAREHOUSESOUTH:I.Data[0].4   // Reserved
           OH_SCAN_WAREHOUSESOUTH:I.Data[0].5   // Reserved
           OH_SCAN_WAREHOUSESOUTH:I.Data[0].6   // Buffer Overflow Error
           OH_SCAN_WAREHOUSESOUTH:I.Data[0].7   // General Error
           OH_SCAN_WAREHOUSESOUTH:I.Data[10]   // ISO/IEC15415 Grade
           OH_SCAN_WAREHOUSESOUTH:I.Data[11]   // Reserved
           OH_SCAN_WAREHOUSESOUTH:I.Data[12]   // AIM DPM Grade
           OH_SCAN_WAREHOUSESOUTH:I.Data[13]   // Reserved
           OH_SCAN_WAREHOUSESOUTH:I.Data[14]   // ISO/IEC15416 Grade
           OH_SCAN_WAREHOUSESOUTH:I.Data[15]   // Reserved
           OH_SCAN_WAREHOUSESOUTH:I.Data[16]   // Read Result Code
           OH_SCAN_WAREHOUSESOUTH:I.Data[17]   // Read Result Code
           OH_SCAN_WAREHOUSESOUTH:I.Data[18]   // Preset Result Code
           OH_SCAN_WAREHOUSESOUTH:I.Data[19]   // Preset Result Code
           OH_SCAN_WAREHOUSESOUTH:I.Data[1].0   // Busy
           OH_SCAN_WAREHOUSESOUTH:I.Data[1].1   // Trigger Busy
           OH_SCAN_WAREHOUSESOUTH:I.Data[1].2   // Lock Busy
           OH_SCAN_WAREHOUSESOUTH:I.Data[1].3   // Mode Busy
           OH_SCAN_WAREHOUSESOUTH:I.Data[1].4   // Error Busy
           OH_SCAN_WAREHOUSESOUTH:I.Data[1].5   // Reserved
           OH_SCAN_WAREHOUSESOUTH:I.Data[1].6   // Ready
           OH_SCAN_WAREHOUSESOUTH:I.Data[1].7   // Reserved
           OH_SCAN_WAREHOUSESOUTH:I.Data[20]   // Register Preset Data Result Code
           OH_SCAN_WAREHOUSESOUTH:I.Data[21]   // Register Preset Data Result Code
           OH_SCAN_WAREHOUSESOUTH:I.Data[22]   // Tune Result Code
           OH_SCAN_WAREHOUSESOUTH:I.Data[23]   // Tune Result Code
           OH_SCAN_WAREHOUSESOUTH:I.Data[24]   // Bload Result Code
           OH_SCAN_WAREHOUSESOUTH:I.Data[25]   // Bload Result Code
           OH_SCAN_WAREHOUSESOUTH:I.Data[26]   // Reserved
           OH_SCAN_WAREHOUSESOUTH:I.Data[27]   // Reserved
           OH_SCAN_WAREHOUSESOUTH:I.Data[28]   // Reserved
           OH_SCAN_WAREHOUSESOUTH:I.Data[29]   // Reserved
           OH_SCAN_WAREHOUSESOUTH:I.Data[2].0   // Read Complete
           OH_SCAN_WAREHOUSESOUTH:I.Data[2].1   // Preset Complete
           OH_SCAN_WAREHOUSESOUTH:I.Data[2].2   // Register Preset Data Complete
           OH_SCAN_WAREHOUSESOUTH:I.Data[2].3   // Tune Complete
           OH_SCAN_WAREHOUSESOUTH:I.Data[2].4   // Bload Complete
           OH_SCAN_WAREHOUSESOUTH:I.Data[2].5   // Reserved
           OH_SCAN_WAREHOUSESOUTH:I.Data[2].6   // Reserved
           OH_SCAN_WAREHOUSESOUTH:I.Data[2].7   // External Request Complete
           OH_SCAN_WAREHOUSESOUTH:I.Data[30]   // External Request Result Code
           OH_SCAN_WAREHOUSESOUTH:I.Data[31]   // External Request Result Code
           OH_SCAN_WAREHOUSESOUTH:I.Data[32]   // General Error Code
           OH_SCAN_WAREHOUSESOUTH:I.Data[33]   // General Error Code
           OH_SCAN_WAREHOUSESOUTH:I.Data[34]   // Slave ID
           OH_SCAN_WAREHOUSESOUTH:I.Data[35]   // Slave ID
           OH_SCAN_WAREHOUSESOUTH:I.Data[36]   // Result Data Ready Count
           OH_SCAN_WAREHOUSESOUTH:I.Data[37]   // Result Data Ready Count
           OH_SCAN_WAREHOUSESOUTH:I.Data[38]   // Result Data Update Count
           OH_SCAN_WAREHOUSESOUTH:I.Data[39]   // Result Data Update Count
           OH_SCAN_WAREHOUSESOUTH:I.Data[3].0   // Read Failure
           OH_SCAN_WAREHOUSESOUTH:I.Data[3].1   // Preset Failure
           OH_SCAN_WAREHOUSESOUTH:I.Data[3].2   // Register Preset Data Failure
           OH_SCAN_WAREHOUSESOUTH:I.Data[3].3   // Tune Failure
           OH_SCAN_WAREHOUSESOUTH:I.Data[3].4   // Bload Failure
           OH_SCAN_WAREHOUSESOUTH:I.Data[3].5   // Reserved
           OH_SCAN_WAREHOUSESOUTH:I.Data[3].6   // Reserved
           OH_SCAN_WAREHOUSESOUTH:I.Data[3].7   // External Request Failure
           OH_SCAN_WAREHOUSESOUTH:I.Data[40]   // Trigger Input Count for Master
           OH_SCAN_WAREHOUSESOUTH:I.Data[41]   // Trigger Input Count for Master
           OH_SCAN_WAREHOUSESOUTH:I.Data[42]   // Result Data Size
           OH_SCAN_WAREHOUSESOUTH:I.Data[43]   // Result Data Size
           OH_SCAN_WAREHOUSESOUTH:I.Data[44]   // Result Data
           OH_SCAN_WAREHOUSESOUTH:I.Data[45]   // Result Data
           OH_SCAN_WAREHOUSESOUTH:I.Data[46]   // Result Data
           OH_SCAN_WAREHOUSESOUTH:I.Data[47]   // Result Data
           OH_SCAN_WAREHOUSESOUTH:I.Data[48]   // Result Data
           OH_SCAN_WAREHOUSESOUTH:I.Data[49]   // Result Data
           OH_SCAN_WAREHOUSESOUTH:I.Data[4].0   // Input 1 Status
           OH_SCAN_WAREHOUSESOUTH:I.Data[4].1   // Input 2 Status
           OH_SCAN_WAREHOUSESOUTH:I.Data[4].2   // Reserved
           OH_SCAN_WAREHOUSESOUTH:I.Data[4].3   // Reserved
           OH_SCAN_WAREHOUSESOUTH:I.Data[4].4   // Output 1 Status
           OH_SCAN_WAREHOUSESOUTH:I.Data[4].5   // Output 2 Status
           OH_SCAN_WAREHOUSESOUTH:I.Data[4].6   // Output 3 Status
           OH_SCAN_WAREHOUSESOUTH:I.Data[4].7   // Reserved
           OH_SCAN_WAREHOUSESOUTH:I.Data[50]   // Result Data
           OH_SCAN_WAREHOUSESOUTH:I.Data[5].0   // Unstable
           OH_SCAN_WAREHOUSESOUTH:I.Data[5].1   // Matching Level Unstable
           OH_SCAN_WAREHOUSESOUTH:I.Data[5].2   // ISO/IEC15415 Unstable
           OH_SCAN_WAREHOUSESOUTH:I.Data[5].3   // AIM DPM Unstable
           OH_SCAN_WAREHOUSESOUTH:I.Data[5].4   // ADE AS9132 Unstable
           OH_SCAN_WAREHOUSESOUTH:I.Data[5].5   // ISO/IEC15416 Unstable
           OH_SCAN_WAREHOUSESOUTH:I.Data[5].6   // Reserved
           OH_SCAN_WAREHOUSESOUTH:I.Data[5].7   // Reserved
           OH_SCAN_WAREHOUSESOUTH:I.Data[6]   // Reserved
           OH_SCAN_WAREHOUSESOUTH:I.Data[7]   // Reserved
           OH_SCAN_WAREHOUSESOUTH:I.Data[8]   // Matching Level
           OH_SCAN_WAREHOUSESOUTH:I.Data[9]   // Reserved
           OH_SCAN_WAREHOUSESOUTH:O.Data[0].0   // Reserved
           OH_SCAN_WAREHOUSESOUTH:O.Data[0].1   // Result Data Latch
           OH_SCAN_WAREHOUSESOUTH:O.Data[0].2   // Reserved
           OH_SCAN_WAREHOUSESOUTH:O.Data[0].3   // Reserved
           OH_SCAN_WAREHOUSESOUTH:O.Data[0].4   // Reserved
           OH_SCAN_WAREHOUSESOUTH:O.Data[0].5   // Reserved
           OH_SCAN_WAREHOUSESOUTH:O.Data[0].6   // Reserved
           OH_SCAN_WAREHOUSESOUTH:O.Data[0].7   // Error Clear
           OH_SCAN_WAREHOUSESOUTH:O.Data[10]   // User Data Size
           OH_SCAN_WAREHOUSESOUTH:O.Data[11]   // User Data Size
           OH_SCAN_WAREHOUSESOUTH:O.Data[12]   // User Data
           OH_SCAN_WAREHOUSESOUTH:O.Data[13]   // User Data
           OH_SCAN_WAREHOUSESOUTH:O.Data[14]   // User Data
           OH_SCAN_WAREHOUSESOUTH:O.Data[15]   // User Data
           OH_SCAN_WAREHOUSESOUTH:O.Data[16]   // User Data
           OH_SCAN_WAREHOUSESOUTH:O.Data[17]   // User Data
           OH_SCAN_WAREHOUSESOUTH:O.Data[1].0   // Read Request
           OH_SCAN_WAREHOUSESOUTH:O.Data[1].1   // Preset Request
           OH_SCAN_WAREHOUSESOUTH:O.Data[1].2   // Register Preset Data Request
           OH_SCAN_WAREHOUSESOUTH:O.Data[1].3   // Tune Request
           OH_SCAN_WAREHOUSESOUTH:O.Data[1].4   // Bload Request
           OH_SCAN_WAREHOUSESOUTH:O.Data[1].5   // Reserved
           OH_SCAN_WAREHOUSESOUTH:O.Data[1].6   // Reserved
           OH_SCAN_WAREHOUSESOUTH:O.Data[1].7   // Reserved
           OH_SCAN_WAREHOUSESOUTH:O.Data[2].0   // Read Complete Clear
           OH_SCAN_WAREHOUSESOUTH:O.Data[2].1   // Preset Complete Clear
           OH_SCAN_WAREHOUSESOUTH:O.Data[2].2   // Register Preset Data Complete Clear
           OH_SCAN_WAREHOUSESOUTH:O.Data[2].3   // Tune Complete Clear
           OH_SCAN_WAREHOUSESOUTH:O.Data[2].4   // Bload Complete Clear
           OH_SCAN_WAREHOUSESOUTH:O.Data[2].5   // Reserved
           OH_SCAN_WAREHOUSESOUTH:O.Data[2].6   // Reserved
           OH_SCAN_WAREHOUSESOUTH:O.Data[2].7   // External Request Complete Clear
           OH_SCAN_WAREHOUSESOUTH:O.Data[3]   // Reserved
           OH_SCAN_WAREHOUSESOUTH:O.Data[4]   // Bank Number
           OH_SCAN_WAREHOUSESOUTH:O.Data[5]   // Bank Number
           OH_SCAN_WAREHOUSESOUTH:O.Data[6]   // Reserved
           OH_SCAN_WAREHOUSESOUTH:O.Data[7]   // Reserved
           OH_SCAN_WAREHOUSESOUTH:O.Data[8]   // Reserved
           OH_SCAN_WAREHOUSESOUTH:O.Data[9]   // Reserved
END_MODULES
